(* Logix 5000 project; controller reports 1756-L63 rev 20.11; software revision 20.04; part 2 of 52 *)

        [93].log_data[7].valid := 1, [93].log_data[8].valid := 1, [93].log_data[9].valid := 1, [93].log_data[10].valid := 1, [93].log_data[11].valid := 1, [93].log_data[12].valid := 1, [93].log_data[13].valid := 1, [93].log_data[14].valid := 1, [93].log_data[15].valid := 1, [93].log_data[16].valid := 1, [93].log_data[17].valid := 1, [93].log_data[18].valid := 1, [93].log_data[19].valid := 1, [93].time.Year := 2023, [93].time.Month := 1, [93].time.Day := 16, [93].time.Hour := 23, [93].time.Minute := 44, [93].time.Second := 59, [94].log_data[0].min := 1.0, [94].log_data[0].max := 1.0, [94].log_data[0].total := 900.0, [94].log_data[0].time := 900.0, [94].log_data[0].minminute := 45, [94].log_data[0].maxminute := 45, [94].log_data[0].valid := 1, [94].log_data[1].valid := 1, [94].log_data[2].valid := 1, [94].log_data[3].valid := 1, [94].log_data[4].valid := 1, [94].log_data[5].valid := 1, [94].log_data[6].valid := 1, [94].log_data[7].valid := 1, [94].log_data[8].valid := 1, [94].log_data[9].valid := 1, [94].log_data[10].valid := 1, [94].log_data[11].valid := 1, [94].log_data[12].valid := 1, [94].log_data[13].valid := 1, [94].log_data[14].valid := 1, [94].log_data[15].valid := 1, [94].log_data[16].valid := 1, [94].log_data[17].valid := 1, [94].log_data[18].valid := 1, [94].log_data[19].valid := 1, [94].time.Year := 2023, [94].time.Month := 1, [94].time.Day := 16, [94].time.Hour := 23, [94].time.Minute := 59, [94].time.Second := 59, [95].log_data[0].min := 1.0, [95].log_data[0].max := 1.0, [95].log_data[0].total := 900.0, [95].log_data[0].time := 900.0, [95].log_data[0].valid := 1, [95].log_data[1].valid := 1, [95].log_data[2].valid := 1, [95].log_data[3].valid := 1, [95].log_data[4].valid := 1,
        [95].log_data[5].valid := 1, [95].log_data[6].valid := 1, [95].log_data[7].valid := 1, [95].log_data[8].valid := 1, [95].log_data[9].valid := 1, [95].log_data[10].valid := 1, [95].log_data[11].valid := 1, [95].log_data[12].valid := 1, [95].log_data[13].valid := 1, [95].log_data[14].valid := 1, [95].log_data[15].valid := 1, [95].log_data[16].valid := 1, [95].log_data[17].valid := 1, [95].log_data[18].valid := 1, [95].log_data[19].valid := 1, [95].time.Year := 2023, [95].time.Month := 1, [95].time.Day := 17, [95].time.Minute := 14, [95].time.Second := 59, [96].log_data[0].min := 1.0, [96].log_data[0].max := 1.0, [96].log_data[0].total := 900.0, [96].log_data[0].time := 900.0, [96].log_data[0].minminute := 15, [96].log_data[0].maxminute := 15, [96].log_data[0].valid := 1, [96].log_data[1].valid := 1, [96].log_data[2].valid := 1, [96].log_data[3].valid := 1, [96].log_data[4].valid := 1, [96].log_data[5].valid := 1, [96].log_data[6].valid := 1, [96].log_data[7].valid := 1, [96].log_data[8].valid := 1, [96].log_data[9].valid := 1, [96].log_data[10].valid := 1, [96].log_data[11].valid := 1, [96].log_data[12].valid := 1, [96].log_data[13].valid := 1, [96].log_data[14].valid := 1, [96].log_data[15].valid := 1, [96].log_data[16].valid := 1, [96].log_data[17].valid := 1, [96].log_data[18].valid := 1, [96].log_data[19].valid := 1, [96].time.Year := 2023, [96].time.Month := 1, [96].time.Day := 17, [96].time.Minute := 29, [96].time.Second := 59, [97].log_data[0].min := 1.0, [97].log_data[0].max := 1.0, [97].log_data[0].total := 900.0, [97].log_data[0].time := 900.0, [97].log_data[0].minminute := 30, [97].log_data[0].maxminute := 30, [97].log_data[0].valid := 1, [97].log_data[1].valid := 1, [97].log_data[2].valid := 1,
        [97].log_data[3].valid := 1, [97].log_data[4].valid := 1, [97].log_data[5].valid := 1, [97].log_data[6].valid := 1, [97].log_data[7].valid := 1, [97].log_data[8].valid := 1, [97].log_data[9].valid := 1, [97].log_data[10].valid := 1, [97].log_data[11].valid := 1, [97].log_data[12].valid := 1, [97].log_data[13].valid := 1, [97].log_data[14].valid := 1, [97].log_data[15].valid := 1, [97].log_data[16].valid := 1, [97].log_data[17].valid := 1, [97].log_data[18].valid := 1, [97].log_data[19].valid := 1, [97].time.Year := 2023, [97].time.Month := 1, [97].time.Day := 17, [97].time.Minute := 44, [97].time.Second := 59, [98].log_data[0].min := 1.0, [98].log_data[0].max := 1.0, [98].log_data[0].total := 900.0, [98].log_data[0].time := 900.0, [98].log_data[0].minminute := 45, [98].log_data[0].maxminute := 45, [98].log_data[0].valid := 1, [98].log_data[1].valid := 1, [98].log_data[2].valid := 1, [98].log_data[3].valid := 1, [98].log_data[4].valid := 1, [98].log_data[5].valid := 1, [98].log_data[6].valid := 1, [98].log_data[7].valid := 1, [98].log_data[8].valid := 1, [98].log_data[9].valid := 1, [98].log_data[10].valid := 1, [98].log_data[11].valid := 1, [98].log_data[12].valid := 1, [98].log_data[13].valid := 1, [98].log_data[14].valid := 1, [98].log_data[15].valid := 1, [98].log_data[16].valid := 1, [98].log_data[17].valid := 1, [98].log_data[18].valid := 1, [98].log_data[19].valid := 1, [98].time.Year := 2023, [98].time.Month := 1, [98].time.Day := 17, [98].time.Minute := 59, [98].time.Second := 59, [99].log_data[0].min := 1.0, [99].log_data[0].max := 1.0, [99].log_data[0].total := 900.0, [99].log_data[0].time := 900.0, [99].log_data[0].valid := 1, [99].log_data[1].valid := 1, [99].log_data[2].valid := 1,
        [99].log_data[3].valid := 1, [99].log_data[4].valid := 1, [99].log_data[5].valid := 1, [99].log_data[6].valid := 1, [99].log_data[7].valid := 1, [99].log_data[8].valid := 1, [99].log_data[9].valid := 1, [99].log_data[10].valid := 1, [99].log_data[11].valid := 1, [99].log_data[12].valid := 1, [99].log_data[13].valid := 1, [99].log_data[14].valid := 1, [99].log_data[15].valid := 1, [99].log_data[16].valid := 1, [99].log_data[17].valid := 1, [99].log_data[18].valid := 1, [99].log_data[19].valid := 1, [99].time.Year := 2023, [99].time.Month := 1, [99].time.Day := 17, [99].time.Hour := 1, [99].time.Minute := 14, [99].time.Second := 59, [100].log_data[0].min := 1.0, [100].log_data[0].max := 1.0, [100].log_data[0].total := 900.0, [100].log_data[0].time := 900.0, [100].log_data[0].minminute := 15, [100].log_data[0].maxminute := 15, [100].log_data[0].valid := 1, [100].log_data[1].valid := 1, [100].log_data[2].valid := 1, [100].log_data[3].valid := 1, [100].log_data[4].valid := 1, [100].log_data[5].valid := 1, [100].log_data[6].valid := 1, [100].log_data[7].valid := 1, [100].log_data[8].valid := 1, [100].log_data[9].valid := 1, [100].log_data[10].valid := 1, [100].log_data[11].valid := 1, [100].log_data[12].valid := 1, [100].log_data[13].valid := 1, [100].log_data[14].valid := 1, [100].log_data[15].valid := 1, [100].log_data[16].valid := 1, [100].log_data[17].valid := 1, [100].log_data[18].valid := 1, [100].log_data[19].valid := 1, [100].time.Year := 2023, [100].time.Month := 1, [100].time.Day := 17, [100].time.Hour := 1, [100].time.Minute := 29, [100].time.Second := 59, [101].log_data[0].min := 1.0, [101].log_data[0].max := 1.0, [101].log_data[0].total := 900.0, [101].log_data[0].time := 900.0, [101].log_data[0].minminute := 30,
        [101].log_data[0].maxminute := 30, [101].log_data[0].valid := 1, [101].log_data[1].valid := 1, [101].log_data[2].valid := 1, [101].log_data[3].valid := 1, [101].log_data[4].valid := 1, [101].log_data[5].valid := 1, [101].log_data[6].valid := 1, [101].log_data[7].valid := 1, [101].log_data[8].valid := 1, [101].log_data[9].valid := 1, [101].log_data[10].valid := 1, [101].log_data[11].valid := 1, [101].log_data[12].valid := 1, [101].log_data[13].valid := 1, [101].log_data[14].valid := 1, [101].log_data[15].valid := 1, [101].log_data[16].valid := 1, [101].log_data[17].valid := 1, [101].log_data[18].valid := 1, [101].log_data[19].valid := 1, [101].time.Year := 2023, [101].time.Month := 1, [101].time.Day := 17, [101].time.Hour := 1, [101].time.Minute := 44, [101].time.Second := 59, [102].log_data[0].min := 1.0, [102].log_data[0].max := 1.0, [102].log_data[0].total := 900.0, [102].log_data[0].time := 900.0, [102].log_data[0].minminute := 45, [102].log_data[0].maxminute := 45, [102].log_data[0].valid := 1, [102].log_data[1].valid := 1, [102].log_data[2].valid := 1, [102].log_data[3].valid := 1, [102].log_data[4].valid := 1, [102].log_data[5].valid := 1, [102].log_data[6].valid := 1, [102].log_data[7].valid := 1, [102].log_data[8].valid := 1, [102].log_data[9].valid := 1, [102].log_data[10].valid := 1, [102].log_data[11].valid := 1, [102].log_data[12].valid := 1, [102].log_data[13].valid := 1, [102].log_data[14].valid := 1, [102].log_data[15].valid := 1, [102].log_data[16].valid := 1, [102].log_data[17].valid := 1, [102].log_data[18].valid := 1, [102].log_data[19].valid := 1, [102].time.Year := 2023, [102].time.Month := 1, [102].time.Day := 17, [102].time.Hour := 1, [102].time.Minute := 59, [102].time.Second := 59, [103].log_data[0].min := 1.0,
        [103].log_data[0].max := 1.0, [103].log_data[0].total := 900.0, [103].log_data[0].time := 900.0, [103].log_data[0].valid := 1, [103].log_data[1].valid := 1, [103].log_data[2].valid := 1, [103].log_data[3].valid := 1, [103].log_data[4].valid := 1, [103].log_data[5].valid := 1, [103].log_data[6].valid := 1, [103].log_data[7].valid := 1, [103].log_data[8].valid := 1, [103].log_data[9].valid := 1, [103].log_data[10].valid := 1, [103].log_data[11].valid := 1, [103].log_data[12].valid := 1, [103].log_data[13].valid := 1, [103].log_data[14].valid := 1, [103].log_data[15].valid := 1, [103].log_data[16].valid := 1, [103].log_data[17].valid := 1, [103].log_data[18].valid := 1, [103].log_data[19].valid := 1, [103].time.Year := 2023, [103].time.Month := 1, [103].time.Day := 17, [103].time.Hour := 2, [103].time.Minute := 14, [103].time.Second := 59, [104].log_data[0].min := 1.0, [104].log_data[0].max := 1.0, [104].log_data[0].total := 900.0, [104].log_data[0].time := 900.0, [104].log_data[0].minminute := 15, [104].log_data[0].maxminute := 15, [104].log_data[0].valid := 1, [104].log_data[1].valid := 1, [104].log_data[2].valid := 1, [104].log_data[3].valid := 1, [104].log_data[4].valid := 1, [104].log_data[5].valid := 1, [104].log_data[6].valid := 1, [104].log_data[7].valid := 1, [104].log_data[8].valid := 1, [104].log_data[9].valid := 1, [104].log_data[10].valid := 1, [104].log_data[11].valid := 1, [104].log_data[12].valid := 1, [104].log_data[13].valid := 1, [104].log_data[14].valid := 1, [104].log_data[15].valid := 1, [104].log_data[16].valid := 1, [104].log_data[17].valid := 1, [104].log_data[18].valid := 1, [104].log_data[19].valid := 1, [104].time.Year := 2023, [104].time.Month := 1, [104].time.Day := 17, [104].time.Hour := 2, [104].time.Minute := 29,
        [104].time.Second := 59, [105].log_data[0].min := 1.0, [105].log_data[0].max := 1.0, [105].log_data[0].total := 900.0, [105].log_data[0].time := 900.0, [105].log_data[0].minminute := 30, [105].log_data[0].maxminute := 30, [105].log_data[0].valid := 1, [105].log_data[1].valid := 1, [105].log_data[2].valid := 1, [105].log_data[3].valid := 1, [105].log_data[4].valid := 1, [105].log_data[5].valid := 1, [105].log_data[6].valid := 1, [105].log_data[7].valid := 1, [105].log_data[8].valid := 1, [105].log_data[9].valid := 1, [105].log_data[10].valid := 1, [105].log_data[11].valid := 1, [105].log_data[12].valid := 1, [105].log_data[13].valid := 1, [105].log_data[14].valid := 1, [105].log_data[15].valid := 1, [105].log_data[16].valid := 1, [105].log_data[17].valid := 1, [105].log_data[18].valid := 1, [105].log_data[19].valid := 1, [105].time.Year := 2023, [105].time.Month := 1, [105].time.Day := 17, [105].time.Hour := 2, [105].time.Minute := 44, [105].time.Second := 59, [106].log_data[0].min := 1.0, [106].log_data[0].max := 1.0, [106].log_data[0].total := 900.0, [106].log_data[0].time := 900.0, [106].log_data[0].minminute := 45, [106].log_data[0].maxminute := 45, [106].log_data[0].valid := 1, [106].log_data[1].valid := 1, [106].log_data[2].valid := 1, [106].log_data[3].valid := 1, [106].log_data[4].valid := 1, [106].log_data[5].valid := 1, [106].log_data[6].valid := 1, [106].log_data[7].valid := 1, [106].log_data[8].valid := 1, [106].log_data[9].valid := 1, [106].log_data[10].valid := 1, [106].log_data[11].valid := 1, [106].log_data[12].valid := 1, [106].log_data[13].valid := 1, [106].log_data[14].valid := 1, [106].log_data[15].valid := 1, [106].log_data[16].valid := 1, [106].log_data[17].valid := 1, [106].log_data[18].valid := 1, [106].log_data[19].valid := 1, [106].time.Year := 2023,
        [106].time.Month := 1, [106].time.Day := 17, [106].time.Hour := 2, [106].time.Minute := 59, [106].time.Second := 59, [107].log_data[0].min := 1.0, [107].log_data[0].max := 1.0, [107].log_data[0].total := 900.0, [107].log_data[0].time := 900.0, [107].log_data[0].valid := 1, [107].log_data[1].valid := 1, [107].log_data[2].valid := 1, [107].log_data[3].valid := 1, [107].log_data[4].valid := 1, [107].log_data[5].valid := 1, [107].log_data[6].valid := 1, [107].log_data[7].valid := 1, [107].log_data[8].valid := 1, [107].log_data[9].valid := 1, [107].log_data[10].valid := 1, [107].log_data[11].valid := 1, [107].log_data[12].valid := 1, [107].log_data[13].valid := 1, [107].log_data[14].valid := 1, [107].log_data[15].valid := 1, [107].log_data[16].valid := 1, [107].log_data[17].valid := 1, [107].log_data[18].valid := 1, [107].log_data[19].valid := 1, [107].time.Year := 2023, [107].time.Month := 1, [107].time.Day := 17, [107].time.Hour := 3, [107].time.Minute := 14, [107].time.Second := 59, [108].log_data[0].min := 1.0, [108].log_data[0].max := 1.0, [108].log_data[0].total := 900.0, [108].log_data[0].time := 900.0, [108].log_data[0].minminute := 15, [108].log_data[0].maxminute := 15, [108].log_data[0].valid := 1, [108].log_data[1].valid := 1, [108].log_data[2].valid := 1, [108].log_data[3].valid := 1, [108].log_data[4].valid := 1, [108].log_data[5].valid := 1, [108].log_data[6].valid := 1, [108].log_data[7].valid := 1, [108].log_data[8].valid := 1, [108].log_data[9].valid := 1, [108].log_data[10].valid := 1, [108].log_data[11].valid := 1, [108].log_data[12].valid := 1, [108].log_data[13].valid := 1, [108].log_data[14].valid := 1, [108].log_data[15].valid := 1, [108].log_data[16].valid := 1, [108].log_data[17].valid := 1, [108].log_data[18].valid := 1,
        [108].log_data[19].valid := 1, [108].time.Year := 2023, [108].time.Month := 1, [108].time.Day := 17, [108].time.Hour := 3, [108].time.Minute := 29, [108].time.Second := 59, [109].log_data[0].min := 1.0, [109].log_data[0].max := 1.0, [109].log_data[0].total := 900.0, [109].log_data[0].time := 900.0, [109].log_data[0].minminute := 30, [109].log_data[0].maxminute := 30, [109].log_data[0].valid := 1, [109].log_data[1].valid := 1, [109].log_data[2].valid := 1, [109].log_data[3].valid := 1, [109].log_data[4].valid := 1, [109].log_data[5].valid := 1, [109].log_data[6].valid := 1, [109].log_data[7].valid := 1, [109].log_data[8].valid := 1, [109].log_data[9].valid := 1, [109].log_data[10].valid := 1, [109].log_data[11].valid := 1, [109].log_data[12].valid := 1, [109].log_data[13].valid := 1, [109].log_data[14].valid := 1, [109].log_data[15].valid := 1, [109].log_data[16].valid := 1, [109].log_data[17].valid := 1, [109].log_data[18].valid := 1, [109].log_data[19].valid := 1, [109].time.Year := 2023, [109].time.Month := 1, [109].time.Day := 17, [109].time.Hour := 3, [109].time.Minute := 44, [109].time.Second := 59, [110].log_data[0].min := 1.0, [110].log_data[0].max := 1.0, [110].log_data[0].total := 900.0, [110].log_data[0].time := 900.0, [110].log_data[0].minminute := 45, [110].log_data[0].maxminute := 45, [110].log_data[0].valid := 1, [110].log_data[1].valid := 1, [110].log_data[2].valid := 1, [110].log_data[3].valid := 1, [110].log_data[4].valid := 1, [110].log_data[5].valid := 1, [110].log_data[6].valid := 1, [110].log_data[7].valid := 1, [110].log_data[8].valid := 1, [110].log_data[9].valid := 1, [110].log_data[10].valid := 1, [110].log_data[11].valid := 1, [110].log_data[12].valid := 1, [110].log_data[13].valid := 1, [110].log_data[14].valid := 1,
        [110].log_data[15].valid := 1, [110].log_data[16].valid := 1, [110].log_data[17].valid := 1, [110].log_data[18].valid := 1, [110].log_data[19].valid := 1, [110].time.Year := 2023, [110].time.Month := 1, [110].time.Day := 17, [110].time.Hour := 3, [110].time.Minute := 59, [110].time.Second := 59, [111].log_data[0].min := 1.0, [111].log_data[0].max := 1.0, [111].log_data[0].total := 900.0, [111].log_data[0].time := 900.0, [111].log_data[0].valid := 1, [111].log_data[1].valid := 1, [111].log_data[2].valid := 1, [111].log_data[3].valid := 1, [111].log_data[4].valid := 1, [111].log_data[5].valid := 1, [111].log_data[6].valid := 1, [111].log_data[7].valid := 1, [111].log_data[8].valid := 1, [111].log_data[9].valid := 1, [111].log_data[10].valid := 1, [111].log_data[11].valid := 1, [111].log_data[12].valid := 1, [111].log_data[13].valid := 1, [111].log_data[14].valid := 1, [111].log_data[15].valid := 1, [111].log_data[16].valid := 1, [111].log_data[17].valid := 1, [111].log_data[18].valid := 1, [111].log_data[19].valid := 1, [111].time.Year := 2023, [111].time.Month := 1, [111].time.Day := 17, [111].time.Hour := 4, [111].time.Minute := 14, [111].time.Second := 59, [112].log_data[0].min := 1.0, [112].log_data[0].max := 1.0, [112].log_data[0].total := 900.0, [112].log_data[0].time := 900.0, [112].log_data[0].minminute := 15, [112].log_data[0].maxminute := 15, [112].log_data[0].valid := 1, [112].log_data[1].valid := 1, [112].log_data[2].valid := 1, [112].log_data[3].valid := 1, [112].log_data[4].valid := 1, [112].log_data[5].valid := 1, [112].log_data[6].valid := 1, [112].log_data[7].valid := 1, [112].log_data[8].valid := 1, [112].log_data[9].valid := 1, [112].log_data[10].valid := 1, [112].log_data[11].valid := 1, [112].log_data[12].valid := 1,
        [112].log_data[13].valid := 1, [112].log_data[14].valid := 1, [112].log_data[15].valid := 1, [112].log_data[16].valid := 1, [112].log_data[17].valid := 1, [112].log_data[18].valid := 1, [112].log_data[19].valid := 1, [112].time.Year := 2023, [112].time.Month := 1, [112].time.Day := 17, [112].time.Hour := 4, [112].time.Minute := 29, [112].time.Second := 59, [113].log_data[0].min := 1.0, [113].log_data[0].max := 1.0, [113].log_data[0].total := 900.0, [113].log_data[0].time := 900.0, [113].log_data[0].minminute := 30, [113].log_data[0].maxminute := 30, [113].log_data[0].valid := 1, [113].log_data[1].valid := 1, [113].log_data[2].valid := 1, [113].log_data[3].valid := 1, [113].log_data[4].valid := 1, [113].log_data[5].valid := 1, [113].log_data[6].valid := 1, [113].log_data[7].valid := 1, [113].log_data[8].valid := 1, [113].log_data[9].valid := 1, [113].log_data[10].valid := 1, [113].log_data[11].valid := 1, [113].log_data[12].valid := 1, [113].log_data[13].valid := 1, [113].log_data[14].valid := 1, [113].log_data[15].valid := 1, [113].log_data[16].valid := 1, [113].log_data[17].valid := 1, [113].log_data[18].valid := 1, [113].log_data[19].valid := 1, [113].time.Year := 2023, [113].time.Month := 1, [113].time.Day := 17, [113].time.Hour := 4, [113].time.Minute := 44, [113].time.Second := 59, [114].log_data[0].min := 1.0, [114].log_data[0].max := 1.0, [114].log_data[0].total := 900.0, [114].log_data[0].time := 900.0, [114].log_data[0].minminute := 45, [114].log_data[0].maxminute := 45, [114].log_data[0].valid := 1, [114].log_data[1].valid := 1, [114].log_data[2].valid := 1, [114].log_data[3].valid := 1, [114].log_data[4].valid := 1, [114].log_data[5].valid := 1, [114].log_data[6].valid := 1, [114].log_data[7].valid := 1, [114].log_data[8].valid := 1,
        [114].log_data[9].valid := 1, [114].log_data[10].valid := 1, [114].log_data[11].valid := 1, [114].log_data[12].valid := 1, [114].log_data[13].valid := 1, [114].log_data[14].valid := 1, [114].log_data[15].valid := 1, [114].log_data[16].valid := 1, [114].log_data[17].valid := 1, [114].log_data[18].valid := 1, [114].log_data[19].valid := 1, [114].time.Year := 2023, [114].time.Month := 1, [114].time.Day := 17, [114].time.Hour := 4, [114].time.Minute := 59, [114].time.Second := 59, [115].log_data[0].min := 1.0, [115].log_data[0].max := 1.0, [115].log_data[0].total := 900.0, [115].log_data[0].time := 900.0, [115].log_data[0].valid := 1, [115].log_data[1].valid := 1, [115].log_data[2].valid := 1, [115].log_data[3].valid := 1, [115].log_data[4].valid := 1, [115].log_data[5].valid := 1, [115].log_data[6].valid := 1, [115].log_data[7].valid := 1, [115].log_data[8].valid := 1, [115].log_data[9].valid := 1, [115].log_data[10].valid := 1, [115].log_data[11].valid := 1, [115].log_data[12].valid := 1, [115].log_data[13].valid := 1, [115].log_data[14].valid := 1, [115].log_data[15].valid := 1, [115].log_data[16].valid := 1, [115].log_data[17].valid := 1, [115].log_data[18].valid := 1, [115].log_data[19].valid := 1, [115].time.Year := 2023, [115].time.Month := 1, [115].time.Day := 17, [115].time.Hour := 5, [115].time.Minute := 14, [115].time.Second := 59, [116].log_data[0].min := 1.0, [116].log_data[0].max := 1.0, [116].log_data[0].total := 900.0, [116].log_data[0].time := 900.0, [116].log_data[0].minminute := 15, [116].log_data[0].maxminute := 15, [116].log_data[0].valid := 1, [116].log_data[1].valid := 1, [116].log_data[2].valid := 1, [116].log_data[3].valid := 1, [116].log_data[4].valid := 1, [116].log_data[5].valid := 1, [116].log_data[6].valid := 1,
        [116].log_data[7].valid := 1, [116].log_data[8].valid := 1, [116].log_data[9].valid := 1, [116].log_data[10].valid := 1, [116].log_data[11].valid := 1, [116].log_data[12].valid := 1, [116].log_data[13].valid := 1, [116].log_data[14].valid := 1, [116].log_data[15].valid := 1, [116].log_data[16].valid := 1, [116].log_data[17].valid := 1, [116].log_data[18].valid := 1, [116].log_data[19].valid := 1, [116].time.Year := 2023, [116].time.Month := 1, [116].time.Day := 17, [116].time.Hour := 5, [116].time.Minute := 29, [116].time.Second := 59, [117].log_data[0].min := 1.0, [117].log_data[0].max := 1.0, [117].log_data[0].total := 900.0, [117].log_data[0].time := 900.0, [117].log_data[0].minminute := 30, [117].log_data[0].maxminute := 30, [117].log_data[0].valid := 1, [117].log_data[1].valid := 1, [117].log_data[2].valid := 1, [117].log_data[3].valid := 1, [117].log_data[4].valid := 1, [117].log_data[5].valid := 1, [117].log_data[6].valid := 1, [117].log_data[7].valid := 1, [117].log_data[8].valid := 1, [117].log_data[9].valid := 1, [117].log_data[10].valid := 1, [117].log_data[11].valid := 1, [117].log_data[12].valid := 1, [117].log_data[13].valid := 1, [117].log_data[14].valid := 1, [117].log_data[15].valid := 1, [117].log_data[16].valid := 1, [117].log_data[17].valid := 1, [117].log_data[18].valid := 1, [117].log_data[19].valid := 1, [117].time.Year := 2023, [117].time.Month := 1, [117].time.Day := 17, [117].time.Hour := 5, [117].time.Minute := 44, [117].time.Second := 59, [118].log_data[0].min := 1.0, [118].log_data[0].max := 1.0, [118].log_data[0].total := 900.0, [118].log_data[0].time := 900.0, [118].log_data[0].minminute := 45, [118].log_data[0].maxminute := 45, [118].log_data[0].valid := 1, [118].log_data[1].valid := 1, [118].log_data[2].valid := 1,
        [118].log_data[3].valid := 1, [118].log_data[4].valid := 1, [118].log_data[5].valid := 1, [118].log_data[6].valid := 1, [118].log_data[7].valid := 1, [118].log_data[8].valid := 1, [118].log_data[9].valid := 1, [118].log_data[10].valid := 1, [118].log_data[11].valid := 1, [118].log_data[12].valid := 1, [118].log_data[13].valid := 1, [118].log_data[14].valid := 1, [118].log_data[15].valid := 1, [118].log_data[16].valid := 1, [118].log_data[17].valid := 1, [118].log_data[18].valid := 1, [118].log_data[19].valid := 1, [118].time.Year := 2023, [118].time.Month := 1, [118].time.Day := 17, [118].time.Hour := 5, [118].time.Minute := 59, [118].time.Second := 59, [119].log_data[0].min := 1.0, [119].log_data[0].max := 1.0, [119].log_data[0].total := 900.0, [119].log_data[0].time := 900.0, [119].log_data[0].valid := 1, [119].log_data[1].valid := 1, [119].log_data[2].valid := 1, [119].log_data[3].valid := 1, [119].log_data[4].valid := 1, [119].log_data[5].valid := 1, [119].log_data[6].valid := 1, [119].log_data[7].valid := 1, [119].log_data[8].valid := 1, [119].log_data[9].valid := 1, [119].log_data[10].valid := 1, [119].log_data[11].valid := 1, [119].log_data[12].valid := 1, [119].log_data[13].valid := 1, [119].log_data[14].valid := 1, [119].log_data[15].valid := 1, [119].log_data[16].valid := 1, [119].log_data[17].valid := 1, [119].log_data[18].valid := 1, [119].log_data[19].valid := 1, [119].time.Year := 2023, [119].time.Month := 1, [119].time.Day := 17, [119].time.Hour := 6, [119].time.Minute := 14, [119].time.Second := 59, [120].log_data[0].min := 1.0, [120].log_data[0].max := 1.0, [120].log_data[0].total := 900.0, [120].log_data[0].time := 900.0, [120].log_data[0].minminute := 15, [120].log_data[0].maxminute := 15, [120].log_data[0].valid := 1,
        [120].log_data[1].valid := 1, [120].log_data[2].valid := 1, [120].log_data[3].valid := 1, [120].log_data[4].valid := 1, [120].log_data[5].valid := 1, [120].log_data[6].valid := 1, [120].log_data[7].valid := 1, [120].log_data[8].valid := 1, [120].log_data[9].valid := 1, [120].log_data[10].valid := 1, [120].log_data[11].valid := 1, [120].log_data[12].valid := 1, [120].log_data[13].valid := 1, [120].log_data[14].valid := 1, [120].log_data[15].valid := 1, [120].log_data[16].valid := 1, [120].log_data[17].valid := 1, [120].log_data[18].valid := 1, [120].log_data[19].valid := 1, [120].time.Year := 2023, [120].time.Month := 1, [120].time.Day := 17, [120].time.Hour := 6, [120].time.Minute := 29, [120].time.Second := 59, [121].log_data[0].min := 1.0, [121].log_data[0].max := 1.0, [121].log_data[0].total := 900.0, [121].log_data[0].time := 900.0, [121].log_data[0].minminute := 30, [121].log_data[0].maxminute := 30, [121].log_data[0].valid := 1, [121].log_data[1].valid := 1, [121].log_data[2].valid := 1, [121].log_data[3].valid := 1, [121].log_data[4].valid := 1, [121].log_data[5].valid := 1, [121].log_data[6].valid := 1, [121].log_data[7].valid := 1, [121].log_data[8].valid := 1, [121].log_data[9].valid := 1, [121].log_data[10].valid := 1, [121].log_data[11].valid := 1, [121].log_data[12].valid := 1, [121].log_data[13].valid := 1, [121].log_data[14].valid := 1, [121].log_data[15].valid := 1, [121].log_data[16].valid := 1, [121].log_data[17].valid := 1, [121].log_data[18].valid := 1, [121].log_data[19].valid := 1, [121].time.Year := 2023, [121].time.Month := 1, [121].time.Day := 17, [121].time.Hour := 6, [121].time.Minute := 44, [121].time.Second := 59, [122].log_data[0].min := 1.0, [122].log_data[0].max := 1.0, [122].log_data[0].total := 900.0,
        [122].log_data[0].time := 900.0, [122].log_data[0].minminute := 45, [122].log_data[0].maxminute := 45, [122].log_data[0].valid := 1, [122].log_data[1].valid := 1, [122].log_data[2].valid := 1, [122].log_data[3].valid := 1, [122].log_data[4].valid := 1, [122].log_data[5].valid := 1, [122].log_data[6].valid := 1, [122].log_data[7].valid := 1, [122].log_data[8].valid := 1, [122].log_data[9].valid := 1, [122].log_data[10].valid := 1, [122].log_data[11].valid := 1, [122].log_data[12].valid := 1, [122].log_data[13].valid := 1, [122].log_data[14].valid := 1, [122].log_data[15].valid := 1, [122].log_data[16].valid := 1, [122].log_data[17].valid := 1, [122].log_data[18].valid := 1, [122].log_data[19].valid := 1, [122].time.Year := 2023, [122].time.Month := 1, [122].time.Day := 17, [122].time.Hour := 6, [122].time.Minute := 59, [122].time.Second := 59, [123].log_data[0].min := 1.0, [123].log_data[0].max := 1.0, [123].log_data[0].total := 900.0, [123].log_data[0].time := 900.0, [123].log_data[0].valid := 1, [123].log_data[1].valid := 1, [123].log_data[2].valid := 1, [123].log_data[3].valid := 1, [123].log_data[4].valid := 1, [123].log_data[5].valid := 1, [123].log_data[6].valid := 1, [123].log_data[7].valid := 1, [123].log_data[8].valid := 1, [123].log_data[9].valid := 1, [123].log_data[10].valid := 1, [123].log_data[11].valid := 1, [123].log_data[12].valid := 1, [123].log_data[13].valid := 1, [123].log_data[14].valid := 1, [123].log_data[15].valid := 1, [123].log_data[16].valid := 1, [123].log_data[17].valid := 1, [123].log_data[18].valid := 1, [123].log_data[19].valid := 1, [123].time.Year := 2023, [123].time.Month := 1, [123].time.Day := 17, [123].time.Hour := 7, [123].time.Minute := 14, [123].time.Second := 59, [124].log_data[0].min := 1.0,
        [124].log_data[0].max := 1.0, [124].log_data[0].total := 900.0, [124].log_data[0].time := 900.0, [124].log_data[0].minminute := 15, [124].log_data[0].maxminute := 15, [124].log_data[0].valid := 1, [124].log_data[1].valid := 1, [124].log_data[2].valid := 1, [124].log_data[3].valid := 1, [124].log_data[4].valid := 1, [124].log_data[5].valid := 1, [124].log_data[6].valid := 1, [124].log_data[7].valid := 1, [124].log_data[8].valid := 1, [124].log_data[9].valid := 1, [124].log_data[10].valid := 1, [124].log_data[11].valid := 1, [124].log_data[12].valid := 1, [124].log_data[13].valid := 1, [124].log_data[14].valid := 1, [124].log_data[15].valid := 1, [124].log_data[16].valid := 1, [124].log_data[17].valid := 1, [124].log_data[18].valid := 1, [124].log_data[19].valid := 1, [124].time.Year := 2023, [124].time.Month := 1, [124].time.Day := 17, [124].time.Hour := 7, [124].time.Minute := 29, [124].time.Second := 59, [125].log_data[0].min := 1.0, [125].log_data[0].max := 1.0, [125].log_data[0].total := 900.0, [125].log_data[0].time := 900.0, [125].log_data[0].minminute := 30, [125].log_data[0].maxminute := 30, [125].log_data[0].valid := 1, [125].log_data[1].valid := 1, [125].log_data[2].valid := 1, [125].log_data[3].valid := 1, [125].log_data[4].valid := 1, [125].log_data[5].valid := 1, [125].log_data[6].valid := 1, [125].log_data[7].valid := 1, [125].log_data[8].valid := 1, [125].log_data[9].valid := 1, [125].log_data[10].valid := 1, [125].log_data[11].valid := 1, [125].log_data[12].valid := 1, [125].log_data[13].valid := 1, [125].log_data[14].valid := 1, [125].log_data[15].valid := 1, [125].log_data[16].valid := 1, [125].log_data[17].valid := 1, [125].log_data[18].valid := 1, [125].log_data[19].valid := 1, [125].time.Year := 2023, [125].time.Month := 1, [125].time.Day := 17,
        [125].time.Hour := 7, [125].time.Minute := 44, [125].time.Second := 59, [126].log_data[0].min := 1.0, [126].log_data[0].max := 1.0, [126].log_data[0].total := 900.0, [126].log_data[0].time := 900.0, [126].log_data[0].minminute := 45, [126].log_data[0].maxminute := 45, [126].log_data[0].valid := 1, [126].log_data[1].valid := 1, [126].log_data[2].valid := 1, [126].log_data[3].valid := 1, [126].log_data[4].valid := 1, [126].log_data[5].valid := 1, [126].log_data[6].valid := 1, [126].log_data[7].valid := 1, [126].log_data[8].valid := 1, [126].log_data[9].valid := 1, [126].log_data[10].valid := 1, [126].log_data[11].valid := 1, [126].log_data[12].valid := 1, [126].log_data[13].valid := 1, [126].log_data[14].valid := 1, [126].log_data[15].valid := 1, [126].log_data[16].valid := 1, [126].log_data[17].valid := 1, [126].log_data[18].valid := 1, [126].log_data[19].valid := 1, [126].time.Year := 2023, [126].time.Month := 1, [126].time.Day := 17, [126].time.Hour := 7, [126].time.Minute := 59, [126].time.Second := 59, [127].log_data[0].min := 1.0, [127].log_data[0].max := 1.0, [127].log_data[0].total := 900.0, [127].log_data[0].time := 900.0, [127].log_data[0].valid := 1, [127].log_data[1].valid := 1, [127].log_data[2].valid := 1, [127].log_data[3].valid := 1, [127].log_data[4].valid := 1, [127].log_data[5].valid := 1, [127].log_data[6].valid := 1, [127].log_data[7].valid := 1, [127].log_data[8].valid := 1, [127].log_data[9].valid := 1, [127].log_data[10].valid := 1, [127].log_data[11].valid := 1, [127].log_data[12].valid := 1, [127].log_data[13].valid := 1, [127].log_data[14].valid := 1, [127].log_data[15].valid := 1, [127].log_data[16].valid := 1, [127].log_data[17].valid := 1, [127].log_data[18].valid := 1, [127].log_data[19].valid := 1, [127].time.Year := 2023,
        [127].time.Month := 1, [127].time.Day := 17, [127].time.Hour := 8, [127].time.Minute := 14, [127].time.Second := 59, [128].log_data[0].min := 1.0, [128].log_data[0].max := 1.0, [128].log_data[0].total := 900.0, [128].log_data[0].time := 900.0, [128].log_data[0].minminute := 15, [128].log_data[0].maxminute := 15, [128].log_data[0].valid := 1, [128].log_data[1].valid := 1, [128].log_data[2].valid := 1, [128].log_data[3].valid := 1, [128].log_data[4].valid := 1, [128].log_data[5].valid := 1, [128].log_data[6].valid := 1, [128].log_data[7].valid := 1, [128].log_data[8].valid := 1, [128].log_data[9].valid := 1, [128].log_data[10].valid := 1, [128].log_data[11].valid := 1, [128].log_data[12].valid := 1, [128].log_data[13].valid := 1, [128].log_data[14].valid := 1, [128].log_data[15].valid := 1, [128].log_data[16].valid := 1, [128].log_data[17].valid := 1, [128].log_data[18].valid := 1, [128].log_data[19].valid := 1, [128].time.Year := 2023, [128].time.Month := 1, [128].time.Day := 17, [128].time.Hour := 8, [128].time.Minute := 29, [128].time.Second := 59, [129].log_data[0].min := 1.0, [129].log_data[0].max := 1.0, [129].log_data[0].total := 900.0, [129].log_data[0].time := 900.0, [129].log_data[0].minminute := 30, [129].log_data[0].maxminute := 30, [129].log_data[0].valid := 1, [129].log_data[1].valid := 1, [129].log_data[2].valid := 1, [129].log_data[3].valid := 1, [129].log_data[4].valid := 1, [129].log_data[5].valid := 1, [129].log_data[6].valid := 1, [129].log_data[7].valid := 1, [129].log_data[8].valid := 1, [129].log_data[9].valid := 1, [129].log_data[10].valid := 1, [129].log_data[11].valid := 1, [129].log_data[12].valid := 1, [129].log_data[13].valid := 1, [129].log_data[14].valid := 1, [129].log_data[15].valid := 1, [129].log_data[16].valid := 1,
        [129].log_data[17].valid := 1, [129].log_data[18].valid := 1, [129].log_data[19].valid := 1, [129].time.Year := 2023, [129].time.Month := 1, [129].time.Day := 17, [129].time.Hour := 8, [129].time.Minute := 44, [129].time.Second := 59, [130].log_data[0].min := 1.0, [130].log_data[0].max := 1.0, [130].log_data[0].total := 900.0, [130].log_data[0].time := 900.0, [130].log_data[0].minminute := 45, [130].log_data[0].maxminute := 45, [130].log_data[0].valid := 1, [130].log_data[1].valid := 1, [130].log_data[2].valid := 1, [130].log_data[3].valid := 1, [130].log_data[4].valid := 1, [130].log_data[5].valid := 1, [130].log_data[6].valid := 1, [130].log_data[7].valid := 1, [130].log_data[8].valid := 1, [130].log_data[9].valid := 1, [130].log_data[10].valid := 1, [130].log_data[11].valid := 1, [130].log_data[12].valid := 1, [130].log_data[13].valid := 1, [130].log_data[14].valid := 1, [130].log_data[15].valid := 1, [130].log_data[16].valid := 1, [130].log_data[17].valid := 1, [130].log_data[18].valid := 1, [130].log_data[19].valid := 1, [130].time.Year := 2023, [130].time.Month := 1, [130].time.Day := 17, [130].time.Hour := 8, [130].time.Minute := 59, [130].time.Second := 59, [131].log_data[0].min := 1.0, [131].log_data[0].max := 1.0, [131].log_data[0].total := 899.5, [131].log_data[0].time := 899.5, [131].log_data[0].valid := 1, [131].log_data[1].valid := 1, [131].log_data[2].valid := 1, [131].log_data[3].valid := 1, [131].log_data[4].valid := 1, [131].log_data[5].valid := 1, [131].log_data[6].valid := 1, [131].log_data[7].valid := 1, [131].log_data[8].valid := 1, [131].log_data[9].valid := 1, [131].log_data[10].valid := 1, [131].log_data[11].valid := 1, [131].log_data[12].valid := 1, [131].log_data[13].valid := 1, [131].log_data[14].valid := 1,
        [131].log_data[15].valid := 1, [131].log_data[16].valid := 1, [131].log_data[17].valid := 1, [131].log_data[18].valid := 1, [131].log_data[19].valid := 1, [131].time.Year := 2023, [131].time.Month := 1, [131].time.Day := 17, [131].time.Hour := 9, [131].time.Minute := 14, [131].time.Second := 59, [132].log_data[0].min := 1.0, [132].log_data[0].max := 1.0, [132].log_data[0].total := 900.0, [132].log_data[0].time := 900.0, [132].log_data[0].minminute := 15, [132].log_data[0].maxminute := 15, [132].log_data[0].valid := 1, [132].log_data[1].valid := 1, [132].log_data[2].valid := 1, [132].log_data[3].valid := 1, [132].log_data[4].valid := 1, [132].log_data[5].valid := 1, [132].log_data[6].valid := 1, [132].log_data[7].valid := 1, [132].log_data[8].valid := 1, [132].log_data[9].valid := 1, [132].log_data[10].valid := 1, [132].log_data[11].valid := 1, [132].log_data[12].valid := 1, [132].log_data[13].valid := 1, [132].log_data[14].valid := 1, [132].log_data[15].valid := 1, [132].log_data[16].valid := 1, [132].log_data[17].valid := 1, [132].log_data[18].valid := 1, [132].log_data[19].valid := 1, [132].time.Year := 2023, [132].time.Month := 1, [132].time.Day := 17, [132].time.Hour := 9, [132].time.Minute := 29, [132].time.Second := 59, [133].log_data[0].min := 1.0, [133].log_data[0].max := 1.0, [133].log_data[0].total := 900.0, [133].log_data[0].time := 900.0, [133].log_data[0].minminute := 30, [133].log_data[0].maxminute := 30, [133].log_data[0].valid := 1, [133].log_data[1].valid := 1, [133].log_data[2].valid := 1, [133].log_data[3].valid := 1, [133].log_data[4].valid := 1, [133].log_data[5].valid := 1, [133].log_data[6].valid := 1, [133].log_data[7].valid := 1, [133].log_data[8].valid := 1, [133].log_data[9].valid := 1, [133].log_data[10].valid := 1,
        [133].log_data[11].valid := 1, [133].log_data[12].valid := 1, [133].log_data[13].valid := 1, [133].log_data[14].valid := 1, [133].log_data[15].valid := 1, [133].log_data[16].valid := 1, [133].log_data[17].valid := 1, [133].log_data[18].valid := 1, [133].log_data[19].valid := 1, [133].time.Year := 2023, [133].time.Month := 1, [133].time.Day := 17, [133].time.Hour := 9, [133].time.Minute := 44, [133].time.Second := 59, [134].log_data[0].min := 1.0, [134].log_data[0].max := 1.0, [134].log_data[0].total := 900.0, [134].log_data[0].time := 900.0, [134].log_data[0].minminute := 45, [134].log_data[0].maxminute := 45, [134].log_data[0].valid := 1, [134].log_data[1].valid := 1, [134].log_data[2].valid := 1, [134].log_data[3].valid := 1, [134].log_data[4].valid := 1, [134].log_data[5].valid := 1, [134].log_data[6].valid := 1, [134].log_data[7].valid := 1, [134].log_data[8].valid := 1, [134].log_data[9].valid := 1, [134].log_data[10].valid := 1, [134].log_data[11].valid := 1, [134].log_data[12].valid := 1, [134].log_data[13].valid := 1, [134].log_data[14].valid := 1, [134].log_data[15].valid := 1, [134].log_data[16].valid := 1, [134].log_data[17].valid := 1, [134].log_data[18].valid := 1, [134].log_data[19].valid := 1, [134].time.Year := 2023, [134].time.Month := 1, [134].time.Day := 17, [134].time.Hour := 9, [134].time.Minute := 59, [134].time.Second := 59, [135].log_data[0].min := 1.0, [135].log_data[0].max := 1.0, [135].log_data[0].total := 900.0, [135].log_data[0].time := 900.0, [135].log_data[0].valid := 1, [135].log_data[1].valid := 1, [135].log_data[2].valid := 1, [135].log_data[3].valid := 1, [135].log_data[4].valid := 1, [135].log_data[5].valid := 1, [135].log_data[6].valid := 1, [135].log_data[7].valid := 1, [135].log_data[8].valid := 1,
        [135].log_data[9].valid := 1, [135].log_data[10].valid := 1, [135].log_data[11].valid := 1, [135].log_data[12].valid := 1, [135].log_data[13].valid := 1, [135].log_data[14].valid := 1, [135].log_data[15].valid := 1, [135].log_data[16].valid := 1, [135].log_data[17].valid := 1, [135].log_data[18].valid := 1, [135].log_data[19].valid := 1, [135].time.Year := 2023, [135].time.Month := 1, [135].time.Day := 17, [135].time.Hour := 10, [135].time.Minute := 14, [135].time.Second := 59, [136].log_data[0].min := 1.0, [136].log_data[0].max := 1.0, [136].log_data[0].total := 900.0, [136].log_data[0].time := 900.0, [136].log_data[0].minminute := 15, [136].log_data[0].maxminute := 15, [136].log_data[0].valid := 1, [136].log_data[1].valid := 1, [136].log_data[2].valid := 1, [136].log_data[3].valid := 1, [136].log_data[4].valid := 1, [136].log_data[5].valid := 1, [136].log_data[6].valid := 1, [136].log_data[7].valid := 1, [136].log_data[8].valid := 1, [136].log_data[9].valid := 1, [136].log_data[10].valid := 1, [136].log_data[11].valid := 1, [136].log_data[12].valid := 1, [136].log_data[13].valid := 1, [136].log_data[14].valid := 1, [136].log_data[15].valid := 1, [136].log_data[16].valid := 1, [136].log_data[17].valid := 1, [136].log_data[18].valid := 1, [136].log_data[19].valid := 1, [136].time.Year := 2023, [136].time.Month := 1, [136].time.Day := 17, [136].time.Hour := 10, [136].time.Minute := 29, [136].time.Second := 59, [137].log_data[0].min := 1.0, [137].log_data[0].max := 1.0, [137].log_data[0].total := 900.0, [137].log_data[0].time := 900.0, [137].log_data[0].minminute := 30, [137].log_data[0].maxminute := 30, [137].log_data[0].valid := 1, [137].log_data[1].valid := 1, [137].log_data[2].valid := 1, [137].log_data[3].valid := 1, [137].log_data[4].valid := 1,
        [137].log_data[5].valid := 1, [137].log_data[6].valid := 1, [137].log_data[7].valid := 1, [137].log_data[8].valid := 1, [137].log_data[9].valid := 1, [137].log_data[10].valid := 1, [137].log_data[11].valid := 1, [137].log_data[12].valid := 1, [137].log_data[13].valid := 1, [137].log_data[14].valid := 1, [137].log_data[15].valid := 1, [137].log_data[16].valid := 1, [137].log_data[17].valid := 1, [137].log_data[18].valid := 1, [137].log_data[19].valid := 1, [137].time.Year := 2023, [137].time.Month := 1, [137].time.Day := 17, [137].time.Hour := 10, [137].time.Minute := 44, [137].time.Second := 59, [138].log_data[0].min := 1.0, [138].log_data[0].max := 1.0, [138].log_data[0].total := 900.0, [138].log_data[0].time := 900.0, [138].log_data[0].minminute := 45, [138].log_data[0].maxminute := 45, [138].log_data[0].valid := 1, [138].log_data[1].valid := 1, [138].log_data[2].valid := 1, [138].log_data[3].valid := 1, [138].log_data[4].valid := 1, [138].log_data[5].valid := 1, [138].log_data[6].valid := 1, [138].log_data[7].valid := 1, [138].log_data[8].valid := 1, [138].log_data[9].valid := 1, [138].log_data[10].valid := 1, [138].log_data[11].valid := 1, [138].log_data[12].valid := 1, [138].log_data[13].valid := 1, [138].log_data[14].valid := 1, [138].log_data[15].valid := 1, [138].log_data[16].valid := 1, [138].log_data[17].valid := 1, [138].log_data[18].valid := 1, [138].log_data[19].valid := 1, [138].time.Year := 2023, [138].time.Month := 1, [138].time.Day := 17, [138].time.Hour := 10, [138].time.Minute := 59, [138].time.Second := 59, [139].log_data[0].min := 1.0, [139].log_data[0].max := 1.0, [139].log_data[0].total := 900.0, [139].log_data[0].time := 900.0, [139].log_data[0].valid := 1, [139].log_data[1].valid := 1, [139].log_data[2].valid := 1,
        [139].log_data[3].valid := 1, [139].log_data[4].valid := 1, [139].log_data[5].valid := 1, [139].log_data[6].valid := 1, [139].log_data[7].valid := 1, [139].log_data[8].valid := 1, [139].log_data[9].valid := 1, [139].log_data[10].valid := 1, [139].log_data[11].valid := 1, [139].log_data[12].valid := 1, [139].log_data[13].valid := 1, [139].log_data[14].valid := 1, [139].log_data[15].valid := 1, [139].log_data[16].valid := 1, [139].log_data[17].valid := 1, [139].log_data[18].valid := 1, [139].log_data[19].valid := 1, [139].time.Year := 2023, [139].time.Month := 1, [139].time.Day := 17, [139].time.Hour := 11, [139].time.Minute := 14, [139].time.Second := 59, [140].log_data[0].min := 1.0, [140].log_data[0].max := 1.0, [140].log_data[0].total := 900.0, [140].log_data[0].time := 900.0, [140].log_data[0].minminute := 15, [140].log_data[0].maxminute := 15, [140].log_data[0].valid := 1, [140].log_data[1].valid := 1, [140].log_data[2].valid := 1, [140].log_data[3].valid := 1, [140].log_data[4].valid := 1, [140].log_data[5].valid := 1, [140].log_data[6].valid := 1, [140].log_data[7].valid := 1, [140].log_data[8].valid := 1, [140].log_data[9].valid := 1, [140].log_data[10].valid := 1, [140].log_data[11].valid := 1, [140].log_data[12].valid := 1, [140].log_data[13].valid := 1, [140].log_data[14].valid := 1, [140].log_data[15].valid := 1, [140].log_data[16].valid := 1, [140].log_data[17].valid := 1, [140].log_data[18].valid := 1, [140].log_data[19].valid := 1, [140].time.Year := 2023, [140].time.Month := 1, [140].time.Day := 17, [140].time.Hour := 11, [140].time.Minute := 29, [140].time.Second := 59, [141].log_data[0].min := 1.0, [141].log_data[0].max := 1.0, [141].log_data[0].total := 900.0, [141].log_data[0].time := 900.0, [141].log_data[0].minminute := 30,
        [141].log_data[0].maxminute := 30, [141].log_data[0].valid := 1, [141].log_data[1].valid := 1, [141].log_data[2].valid := 1, [141].log_data[3].valid := 1, [141].log_data[4].valid := 1, [141].log_data[5].valid := 1, [141].log_data[6].valid := 1, [141].log_data[7].valid := 1, [141].log_data[8].valid := 1, [141].log_data[9].valid := 1, [141].log_data[10].valid := 1, [141].log_data[11].valid := 1, [141].log_data[12].valid := 1, [141].log_data[13].valid := 1, [141].log_data[14].valid := 1, [141].log_data[15].valid := 1, [141].log_data[16].valid := 1, [141].log_data[17].valid := 1, [141].log_data[18].valid := 1, [141].log_data[19].valid := 1, [141].time.Year := 2023, [141].time.Month := 1, [141].time.Day := 17, [141].time.Hour := 11, [141].time.Minute := 44, [141].time.Second := 59, [142].log_data[0].min := 1.0, [142].log_data[0].max := 1.0, [142].log_data[0].total := 900.0, [142].log_data[0].time := 900.0, [142].log_data[0].minminute := 45, [142].log_data[0].maxminute := 45, [142].log_data[0].valid := 1, [142].log_data[1].valid := 1, [142].log_data[2].valid := 1, [142].log_data[3].valid := 1, [142].log_data[4].valid := 1, [142].log_data[5].valid := 1, [142].log_data[6].valid := 1, [142].log_data[7].valid := 1, [142].log_data[8].valid := 1, [142].log_data[9].valid := 1, [142].log_data[10].valid := 1, [142].log_data[11].valid := 1, [142].log_data[12].valid := 1, [142].log_data[13].valid := 1, [142].log_data[14].valid := 1, [142].log_data[15].valid := 1, [142].log_data[16].valid := 1, [142].log_data[17].valid := 1, [142].log_data[18].valid := 1, [142].log_data[19].valid := 1, [142].time.Year := 2023, [142].time.Month := 1, [142].time.Day := 17, [142].time.Hour := 11, [142].time.Minute := 59, [142].time.Second := 59, [143].log_data[0].min := 1.0,
        [143].log_data[0].max := 1.0, [143].log_data[0].total := 900.0, [143].log_data[0].time := 900.0, [143].log_data[0].valid := 1, [143].log_data[1].valid := 1, [143].log_data[2].valid := 1, [143].log_data[3].valid := 1, [143].log_data[4].valid := 1, [143].log_data[5].valid := 1, [143].log_data[6].valid := 1, [143].log_data[7].valid := 1, [143].log_data[8].valid := 1, [143].log_data[9].valid := 1, [143].log_data[10].valid := 1, [143].log_data[11].valid := 1, [143].log_data[12].valid := 1, [143].log_data[13].valid := 1, [143].log_data[14].valid := 1, [143].log_data[15].valid := 1, [143].log_data[16].valid := 1, [143].log_data[17].valid := 1, [143].log_data[18].valid := 1, [143].log_data[19].valid := 1, [143].time.Year := 2023, [143].time.Month := 1, [143].time.Day := 17, [143].time.Hour := 12, [143].time.Minute := 14, [143].time.Second := 59, [144].log_data[0].min := 1.0, [144].log_data[0].max := 1.0, [144].log_data[0].total := 900.0, [144].log_data[0].time := 900.0, [144].log_data[0].minminute := 15, [144].log_data[0].maxminute := 15, [144].log_data[0].valid := 1, [144].log_data[1].valid := 1, [144].log_data[2].valid := 1, [144].log_data[3].valid := 1, [144].log_data[4].valid := 1, [144].log_data[5].valid := 1, [144].log_data[6].valid := 1, [144].log_data[7].valid := 1, [144].log_data[8].valid := 1, [144].log_data[9].valid := 1, [144].log_data[10].valid := 1, [144].log_data[11].valid := 1, [144].log_data[12].valid := 1, [144].log_data[13].valid := 1, [144].log_data[14].valid := 1, [144].log_data[15].valid := 1, [144].log_data[16].valid := 1, [144].log_data[17].valid := 1, [144].log_data[18].valid := 1, [144].log_data[19].valid := 1, [144].time.Year := 2023, [144].time.Month := 1, [144].time.Day := 17, [144].time.Hour := 12, [144].time.Minute := 29,
        [144].time.Second := 59, [145].log_data[0].min := 1.0, [145].log_data[0].max := 1.0, [145].log_data[0].total := 900.0, [145].log_data[0].time := 900.0, [145].log_data[0].minminute := 30, [145].log_data[0].maxminute := 30, [145].log_data[0].valid := 1, [145].log_data[1].valid := 1, [145].log_data[2].valid := 1, [145].log_data[3].valid := 1, [145].log_data[4].valid := 1, [145].log_data[5].valid := 1, [145].log_data[6].valid := 1, [145].log_data[7].valid := 1, [145].log_data[8].valid := 1, [145].log_data[9].valid := 1, [145].log_data[10].valid := 1, [145].log_data[11].valid := 1, [145].log_data[12].valid := 1, [145].log_data[13].valid := 1, [145].log_data[14].valid := 1, [145].log_data[15].valid := 1, [145].log_data[16].valid := 1, [145].log_data[17].valid := 1, [145].log_data[18].valid := 1, [145].log_data[19].valid := 1, [145].time.Year := 2023, [145].time.Month := 1, [145].time.Day := 17, [145].time.Hour := 12, [145].time.Minute := 44, [145].time.Second := 59, [146].log_data[0].min := 1.0, [146].log_data[0].max := 1.0, [146].log_data[0].total := 900.0, [146].log_data[0].time := 900.0, [146].log_data[0].minminute := 45, [146].log_data[0].maxminute := 45, [146].log_data[0].valid := 1, [146].log_data[1].valid := 1, [146].log_data[2].valid := 1, [146].log_data[3].valid := 1, [146].log_data[4].valid := 1, [146].log_data[5].valid := 1, [146].log_data[6].valid := 1, [146].log_data[7].valid := 1, [146].log_data[8].valid := 1, [146].log_data[9].valid := 1, [146].log_data[10].valid := 1, [146].log_data[11].valid := 1, [146].log_data[12].valid := 1, [146].log_data[13].valid := 1, [146].log_data[14].valid := 1, [146].log_data[15].valid := 1, [146].log_data[16].valid := 1, [146].log_data[17].valid := 1, [146].log_data[18].valid := 1, [146].log_data[19].valid := 1, [146].time.Year := 2023,
        [146].time.Month := 1, [146].time.Day := 17, [146].time.Hour := 12, [146].time.Minute := 59, [146].time.Second := 59, [147].log_data[0].min := 1.0, [147].log_data[0].max := 1.0, [147].log_data[0].total := 900.0, [147].log_data[0].time := 900.0, [147].log_data[0].valid := 1, [147].log_data[1].valid := 1, [147].log_data[2].valid := 1, [147].log_data[3].valid := 1, [147].log_data[4].valid := 1, [147].log_data[5].valid := 1, [147].log_data[6].valid := 1, [147].log_data[7].valid := 1, [147].log_data[8].valid := 1, [147].log_data[9].valid := 1, [147].log_data[10].valid := 1, [147].log_data[11].valid := 1, [147].log_data[12].valid := 1, [147].log_data[13].valid := 1, [147].log_data[14].valid := 1, [147].log_data[15].valid := 1, [147].log_data[16].valid := 1, [147].log_data[17].valid := 1, [147].log_data[18].valid := 1, [147].log_data[19].valid := 1, [147].time.Year := 2023, [147].time.Month := 1, [147].time.Day := 17, [147].time.Hour := 13, [147].time.Minute := 14, [147].time.Second := 59, [148].log_data[0].min := 1.0, [148].log_data[0].max := 1.0, [148].log_data[0].total := 900.0, [148].log_data[0].time := 900.0, [148].log_data[0].minminute := 15, [148].log_data[0].maxminute := 15, [148].log_data[0].valid := 1, [148].log_data[1].valid := 1, [148].log_data[2].valid := 1, [148].log_data[3].valid := 1, [148].log_data[4].valid := 1, [148].log_data[5].valid := 1, [148].log_data[6].valid := 1, [148].log_data[7].valid := 1, [148].log_data[8].valid := 1, [148].log_data[9].valid := 1, [148].log_data[10].valid := 1, [148].log_data[11].valid := 1, [148].log_data[12].valid := 1, [148].log_data[13].valid := 1, [148].log_data[14].valid := 1, [148].log_data[15].valid := 1, [148].log_data[16].valid := 1, [148].log_data[17].valid := 1, [148].log_data[18].valid := 1,
        [148].log_data[19].valid := 1, [148].time.Year := 2023, [148].time.Month := 1, [148].time.Day := 17, [148].time.Hour := 13, [148].time.Minute := 29, [148].time.Second := 59, [149].log_data[0].min := 1.0, [149].log_data[0].max := 1.0, [149].log_data[0].total := 900.0, [149].log_data[0].time := 900.0, [149].log_data[0].minminute := 30, [149].log_data[0].maxminute := 30, [149].log_data[0].valid := 1, [149].log_data[1].valid := 1, [149].log_data[2].valid := 1, [149].log_data[3].valid := 1, [149].log_data[4].valid := 1, [149].log_data[5].valid := 1, [149].log_data[6].valid := 1, [149].log_data[7].valid := 1, [149].log_data[8].valid := 1, [149].log_data[9].valid := 1, [149].log_data[10].valid := 1, [149].log_data[11].valid := 1, [149].log_data[12].valid := 1, [149].log_data[13].valid := 1, [149].log_data[14].valid := 1, [149].log_data[15].valid := 1, [149].log_data[16].valid := 1, [149].log_data[17].valid := 1, [149].log_data[18].valid := 1, [149].log_data[19].valid := 1, [149].time.Year := 2023, [149].time.Month := 1, [149].time.Day := 17, [149].time.Hour := 13, [149].time.Minute := 44, [149].time.Second := 59, [150].log_data[0].min := 1.0, [150].log_data[0].max := 1.0, [150].log_data[0].total := 900.0, [150].log_data[0].time := 900.0, [150].log_data[0].minminute := 45, [150].log_data[0].maxminute := 45, [150].log_data[0].valid := 1, [150].log_data[1].valid := 1, [150].log_data[2].valid := 1, [150].log_data[3].valid := 1, [150].log_data[4].valid := 1, [150].log_data[5].valid := 1, [150].log_data[6].valid := 1, [150].log_data[7].valid := 1, [150].log_data[8].valid := 1, [150].log_data[9].valid := 1, [150].log_data[10].valid := 1, [150].log_data[11].valid := 1, [150].log_data[12].valid := 1, [150].log_data[13].valid := 1, [150].log_data[14].valid := 1,
        [150].log_data[15].valid := 1, [150].log_data[16].valid := 1, [150].log_data[17].valid := 1, [150].log_data[18].valid := 1, [150].log_data[19].valid := 1, [150].time.Year := 2023, [150].time.Month := 1, [150].time.Day := 17, [150].time.Hour := 13, [150].time.Minute := 59, [150].time.Second := 59, [151].log_data[0].min := 1.0, [151].log_data[0].max := 1.0, [151].log_data[0].total := 900.0, [151].log_data[0].time := 900.0, [151].log_data[0].valid := 1, [151].log_data[1].valid := 1, [151].log_data[2].valid := 1, [151].log_data[3].valid := 1, [151].log_data[4].valid := 1, [151].log_data[5].valid := 1, [151].log_data[6].valid := 1, [151].log_data[7].valid := 1, [151].log_data[8].valid := 1, [151].log_data[9].valid := 1, [151].log_data[10].valid := 1, [151].log_data[11].valid := 1, [151].log_data[12].valid := 1, [151].log_data[13].valid := 1, [151].log_data[14].valid := 1, [151].log_data[15].valid := 1, [151].log_data[16].valid := 1, [151].log_data[17].valid := 1, [151].log_data[18].valid := 1, [151].log_data[19].valid := 1, [151].time.Year := 2023, [151].time.Month := 1, [151].time.Day := 17, [151].time.Hour := 14, [151].time.Minute := 14, [151].time.Second := 59, [152].log_data[0].min := 1.0, [152].log_data[0].max := 1.0, [152].log_data[0].total := 900.0, [152].log_data[0].time := 900.0, [152].log_data[0].minminute := 15, [152].log_data[0].maxminute := 15, [152].log_data[0].valid := 1, [152].log_data[1].valid := 1, [152].log_data[2].valid := 1, [152].log_data[3].valid := 1, [152].log_data[4].valid := 1, [152].log_data[5].valid := 1, [152].log_data[6].valid := 1, [152].log_data[7].valid := 1, [152].log_data[8].valid := 1, [152].log_data[9].valid := 1, [152].log_data[10].valid := 1, [152].log_data[11].valid := 1, [152].log_data[12].valid := 1,
        [152].log_data[13].valid := 1, [152].log_data[14].valid := 1, [152].log_data[15].valid := 1, [152].log_data[16].valid := 1, [152].log_data[17].valid := 1, [152].log_data[18].valid := 1, [152].log_data[19].valid := 1, [152].time.Year := 2023, [152].time.Month := 1, [152].time.Day := 17, [152].time.Hour := 14, [152].time.Minute := 29, [152].time.Second := 59, [153].log_data[0].min := 1.0, [153].log_data[0].max := 1.0, [153].log_data[0].total := 900.0, [153].log_data[0].time := 900.0, [153].log_data[0].minminute := 30, [153].log_data[0].maxminute := 30, [153].log_data[0].valid := 1, [153].log_data[1].valid := 1, [153].log_data[2].valid := 1, [153].log_data[3].valid := 1, [153].log_data[4].valid := 1, [153].log_data[5].valid := 1, [153].log_data[6].valid := 1, [153].log_data[7].valid := 1, [153].log_data[8].valid := 1, [153].log_data[9].valid := 1, [153].log_data[10].valid := 1, [153].log_data[11].valid := 1, [153].log_data[12].valid := 1, [153].log_data[13].valid := 1, [153].log_data[14].valid := 1, [153].log_data[15].valid := 1, [153].log_data[16].valid := 1, [153].log_data[17].valid := 1, [153].log_data[18].valid := 1, [153].log_data[19].valid := 1, [153].time.Year := 2023, [153].time.Month := 1, [153].time.Day := 17, [153].time.Hour := 14, [153].time.Minute := 44, [153].time.Second := 59, [154].log_data[0].min := 1.0, [154].log_data[0].max := 1.0, [154].log_data[0].total := 900.0, [154].log_data[0].time := 900.0, [154].log_data[0].minminute := 45, [154].log_data[0].maxminute := 45, [154].log_data[0].valid := 1, [154].log_data[1].valid := 1, [154].log_data[2].valid := 1, [154].log_data[3].valid := 1, [154].log_data[4].valid := 1, [154].log_data[5].valid := 1, [154].log_data[6].valid := 1, [154].log_data[7].valid := 1, [154].log_data[8].valid := 1,
        [154].log_data[9].valid := 1, [154].log_data[10].valid := 1, [154].log_data[11].valid := 1, [154].log_data[12].valid := 1, [154].log_data[13].valid := 1, [154].log_data[14].valid := 1, [154].log_data[15].valid := 1, [154].log_data[16].valid := 1, [154].log_data[17].valid := 1, [154].log_data[18].valid := 1, [154].log_data[19].valid := 1, [154].time.Year := 2023, [154].time.Month := 1, [154].time.Day := 17, [154].time.Hour := 14, [154].time.Minute := 59, [154].time.Second := 59, [155].log_data[0].min := 1.0, [155].log_data[0].max := 1.0, [155].log_data[0].total := 900.0, [155].log_data[0].time := 900.0, [155].log_data[0].valid := 1, [155].log_data[1].valid := 1, [155].log_data[2].valid := 1, [155].log_data[3].valid := 1, [155].log_data[4].valid := 1, [155].log_data[5].valid := 1, [155].log_data[6].valid := 1, [155].log_data[7].valid := 1, [155].log_data[8].valid := 1, [155].log_data[9].valid := 1, [155].log_data[10].valid := 1, [155].log_data[11].valid := 1, [155].log_data[12].valid := 1, [155].log_data[13].valid := 1, [155].log_data[14].valid := 1, [155].log_data[15].valid := 1, [155].log_data[16].valid := 1, [155].log_data[17].valid := 1, [155].log_data[18].valid := 1, [155].log_data[19].valid := 1, [155].time.Year := 2023, [155].time.Month := 1, [155].time.Day := 17, [155].time.Hour := 15, [155].time.Minute := 14, [155].time.Second := 59, [156].log_data[0].min := 1.0, [156].log_data[0].max := 1.0, [156].log_data[0].total := 900.0, [156].log_data[0].time := 900.0, [156].log_data[0].minminute := 15, [156].log_data[0].maxminute := 15, [156].log_data[0].valid := 1, [156].log_data[1].valid := 1, [156].log_data[2].valid := 1, [156].log_data[3].valid := 1, [156].log_data[4].valid := 1, [156].log_data[5].valid := 1, [156].log_data[6].valid := 1,
        [156].log_data[7].valid := 1, [156].log_data[8].valid := 1, [156].log_data[9].valid := 1, [156].log_data[10].valid := 1, [156].log_data[11].valid := 1, [156].log_data[12].valid := 1, [156].log_data[13].valid := 1, [156].log_data[14].valid := 1, [156].log_data[15].valid := 1, [156].log_data[16].valid := 1, [156].log_data[17].valid := 1, [156].log_data[18].valid := 1, [156].log_data[19].valid := 1, [156].time.Year := 2023, [156].time.Month := 1, [156].time.Day := 17, [156].time.Hour := 15, [156].time.Minute := 29, [156].time.Second := 59, [157].log_data[0].min := 1.0, [157].log_data[0].max := 1.0, [157].log_data[0].total := 900.0, [157].log_data[0].time := 900.0, [157].log_data[0].minminute := 30, [157].log_data[0].maxminute := 30, [157].log_data[0].valid := 1, [157].log_data[1].valid := 1, [157].log_data[2].valid := 1, [157].log_data[3].valid := 1, [157].log_data[4].valid := 1, [157].log_data[5].valid := 1, [157].log_data[6].valid := 1, [157].log_data[7].valid := 1, [157].log_data[8].valid := 1, [157].log_data[9].valid := 1, [157].log_data[10].valid := 1, [157].log_data[11].valid := 1, [157].log_data[12].valid := 1, [157].log_data[13].valid := 1, [157].log_data[14].valid := 1, [157].log_data[15].valid := 1, [157].log_data[16].valid := 1, [157].log_data[17].valid := 1, [157].log_data[18].valid := 1, [157].log_data[19].valid := 1, [157].time.Year := 2023, [157].time.Month := 1, [157].time.Day := 17, [157].time.Hour := 15, [157].time.Minute := 44, [157].time.Second := 59, [158].log_data[0].min := 1.0, [158].log_data[0].max := 1.0, [158].log_data[0].total := 900.0, [158].log_data[0].time := 900.0, [158].log_data[0].minminute := 45, [158].log_data[0].maxminute := 45, [158].log_data[0].valid := 1, [158].log_data[1].valid := 1, [158].log_data[2].valid := 1,
        [158].log_data[3].valid := 1, [158].log_data[4].valid := 1, [158].log_data[5].valid := 1, [158].log_data[6].valid := 1, [158].log_data[7].valid := 1, [158].log_data[8].valid := 1, [158].log_data[9].valid := 1, [158].log_data[10].valid := 1, [158].log_data[11].valid := 1, [158].log_data[12].valid := 1, [158].log_data[13].valid := 1, [158].log_data[14].valid := 1, [158].log_data[15].valid := 1, [158].log_data[16].valid := 1, [158].log_data[17].valid := 1, [158].log_data[18].valid := 1, [158].log_data[19].valid := 1, [158].time.Year := 2023, [158].time.Month := 1, [158].time.Day := 17, [158].time.Hour := 15, [158].time.Minute := 59, [158].time.Second := 59, [159].log_data[0].min := 1.0, [159].log_data[0].max := 1.0, [159].log_data[0].total := 900.0, [159].log_data[0].time := 900.0, [159].log_data[0].valid := 1, [159].log_data[1].valid := 1, [159].log_data[2].valid := 1, [159].log_data[3].valid := 1, [159].log_data[4].valid := 1, [159].log_data[5].valid := 1, [159].log_data[6].valid := 1, [159].log_data[7].valid := 1, [159].log_data[8].valid := 1, [159].log_data[9].valid := 1, [159].log_data[10].valid := 1, [159].log_data[11].valid := 1, [159].log_data[12].valid := 1, [159].log_data[13].valid := 1, [159].log_data[14].valid := 1, [159].log_data[15].valid := 1, [159].log_data[16].valid := 1, [159].log_data[17].valid := 1, [159].log_data[18].valid := 1, [159].log_data[19].valid := 1, [159].time.Year := 2023, [159].time.Month := 1, [159].time.Day := 17, [159].time.Hour := 16, [159].time.Minute := 14, [159].time.Second := 59, [160].log_data[0].min := 1.0, [160].log_data[0].max := 1.0, [160].log_data[0].total := 900.0, [160].log_data[0].time := 900.0, [160].log_data[0].minminute := 15, [160].log_data[0].maxminute := 15, [160].log_data[0].valid := 1,
        [160].log_data[1].valid := 1, [160].log_data[2].valid := 1, [160].log_data[3].valid := 1, [160].log_data[4].valid := 1, [160].log_data[5].valid := 1, [160].log_data[6].valid := 1, [160].log_data[7].valid := 1, [160].log_data[8].valid := 1, [160].log_data[9].valid := 1, [160].log_data[10].valid := 1, [160].log_data[11].valid := 1, [160].log_data[12].valid := 1, [160].log_data[13].valid := 1, [160].log_data[14].valid := 1, [160].log_data[15].valid := 1, [160].log_data[16].valid := 1, [160].log_data[17].valid := 1, [160].log_data[18].valid := 1, [160].log_data[19].valid := 1, [160].time.Year := 2023, [160].time.Month := 1, [160].time.Day := 17, [160].time.Hour := 16, [160].time.Minute := 29, [160].time.Second := 59, [161].log_data[0].min := 1.0, [161].log_data[0].max := 1.0, [161].log_data[0].total := 900.0, [161].log_data[0].time := 900.0, [161].log_data[0].minminute := 30, [161].log_data[0].maxminute := 30, [161].log_data[0].valid := 1, [161].log_data[1].valid := 1, [161].log_data[2].valid := 1, [161].log_data[3].valid := 1, [161].log_data[4].valid := 1, [161].log_data[5].valid := 1, [161].log_data[6].valid := 1, [161].log_data[7].valid := 1, [161].log_data[8].valid := 1, [161].log_data[9].valid := 1, [161].log_data[10].valid := 1, [161].log_data[11].valid := 1, [161].log_data[12].valid := 1, [161].log_data[13].valid := 1, [161].log_data[14].valid := 1, [161].log_data[15].valid := 1, [161].log_data[16].valid := 1, [161].log_data[17].valid := 1, [161].log_data[18].valid := 1, [161].log_data[19].valid := 1, [161].time.Year := 2023, [161].time.Month := 1, [161].time.Day := 17, [161].time.Hour := 16, [161].time.Minute := 44, [161].time.Second := 59, [162].log_data[0].min := 1.0, [162].log_data[0].max := 1.0, [162].log_data[0].total := 900.0,
        [162].log_data[0].time := 900.0, [162].log_data[0].minminute := 45, [162].log_data[0].maxminute := 45, [162].log_data[0].valid := 1, [162].log_data[1].valid := 1, [162].log_data[2].valid := 1, [162].log_data[3].valid := 1, [162].log_data[4].valid := 1, [162].log_data[5].valid := 1, [162].log_data[6].valid := 1, [162].log_data[7].valid := 1, [162].log_data[8].valid := 1, [162].log_data[9].valid := 1, [162].log_data[10].valid := 1, [162].log_data[11].valid := 1, [162].log_data[12].valid := 1, [162].log_data[13].valid := 1, [162].log_data[14].valid := 1, [162].log_data[15].valid := 1, [162].log_data[16].valid := 1, [162].log_data[17].valid := 1, [162].log_data[18].valid := 1, [162].log_data[19].valid := 1, [162].time.Year := 2023, [162].time.Month := 1, [162].time.Day := 17, [162].time.Hour := 16, [162].time.Minute := 59, [162].time.Second := 59, [163].log_data[0].min := 1.0, [163].log_data[0].max := 1.0, [163].log_data[0].total := 900.0, [163].log_data[0].time := 900.0, [163].log_data[0].valid := 1, [163].log_data[1].valid := 1, [163].log_data[2].valid := 1, [163].log_data[3].valid := 1, [163].log_data[4].valid := 1, [163].log_data[5].valid := 1, [163].log_data[6].valid := 1, [163].log_data[7].valid := 1, [163].log_data[8].valid := 1, [163].log_data[9].valid := 1, [163].log_data[10].valid := 1, [163].log_data[11].valid := 1, [163].log_data[12].valid := 1, [163].log_data[13].valid := 1, [163].log_data[14].valid := 1, [163].log_data[15].valid := 1, [163].log_data[16].valid := 1, [163].log_data[17].valid := 1, [163].log_data[18].valid := 1, [163].log_data[19].valid := 1, [163].time.Year := 2023, [163].time.Month := 1, [163].time.Day := 17, [163].time.Hour := 17, [163].time.Minute := 14, [163].time.Second := 59, [164].log_data[0].min := 1.0,
        [164].log_data[0].max := 1.0, [164].log_data[0].total := 900.0, [164].log_data[0].time := 900.0, [164].log_data[0].minminute := 15, [164].log_data[0].maxminute := 15, [164].log_data[0].valid := 1, [164].log_data[1].valid := 1, [164].log_data[2].valid := 1, [164].log_data[3].valid := 1, [164].log_data[4].valid := 1, [164].log_data[5].valid := 1, [164].log_data[6].valid := 1, [164].log_data[7].valid := 1, [164].log_data[8].valid := 1, [164].log_data[9].valid := 1, [164].log_data[10].valid := 1, [164].log_data[11].valid := 1, [164].log_data[12].valid := 1, [164].log_data[13].valid := 1, [164].log_data[14].valid := 1, [164].log_data[15].valid := 1, [164].log_data[16].valid := 1, [164].log_data[17].valid := 1, [164].log_data[18].valid := 1, [164].log_data[19].valid := 1, [164].time.Year := 2023, [164].time.Month := 1, [164].time.Day := 17, [164].time.Hour := 17, [164].time.Minute := 29, [164].time.Second := 59, [165].log_data[0].min := 1.0, [165].log_data[0].max := 1.0, [165].log_data[0].total := 900.0, [165].log_data[0].time := 900.0, [165].log_data[0].minminute := 30, [165].log_data[0].maxminute := 30, [165].log_data[0].valid := 1, [165].log_data[1].valid := 1, [165].log_data[2].valid := 1, [165].log_data[3].valid := 1, [165].log_data[4].valid := 1, [165].log_data[5].valid := 1, [165].log_data[6].valid := 1, [165].log_data[7].valid := 1, [165].log_data[8].valid := 1, [165].log_data[9].valid := 1, [165].log_data[10].valid := 1, [165].log_data[11].valid := 1, [165].log_data[12].valid := 1, [165].log_data[13].valid := 1, [165].log_data[14].valid := 1, [165].log_data[15].valid := 1, [165].log_data[16].valid := 1, [165].log_data[17].valid := 1, [165].log_data[18].valid := 1, [165].log_data[19].valid := 1, [165].time.Year := 2023, [165].time.Month := 1, [165].time.Day := 17,
        [165].time.Hour := 17, [165].time.Minute := 44, [165].time.Second := 59, [166].log_data[0].min := 1.0, [166].log_data[0].max := 1.0, [166].log_data[0].total := 900.0, [166].log_data[0].time := 900.0, [166].log_data[0].minminute := 45, [166].log_data[0].maxminute := 45, [166].log_data[0].valid := 1, [166].log_data[1].valid := 1, [166].log_data[2].valid := 1, [166].log_data[3].valid := 1, [166].log_data[4].valid := 1, [166].log_data[5].valid := 1, [166].log_data[6].valid := 1, [166].log_data[7].valid := 1, [166].log_data[8].valid := 1, [166].log_data[9].valid := 1, [166].log_data[10].valid := 1, [166].log_data[11].valid := 1, [166].log_data[12].valid := 1, [166].log_data[13].valid := 1, [166].log_data[14].valid := 1, [166].log_data[15].valid := 1, [166].log_data[16].valid := 1, [166].log_data[17].valid := 1, [166].log_data[18].valid := 1, [166].log_data[19].valid := 1, [166].time.Year := 2023, [166].time.Month := 1, [166].time.Day := 17, [166].time.Hour := 17, [166].time.Minute := 59, [166].time.Second := 59, [167].log_data[0].min := 1.0, [167].log_data[0].max := 1.0, [167].log_data[0].total := 900.0, [167].log_data[0].time := 900.0, [167].log_data[0].valid := 1, [167].log_data[1].valid := 1, [167].log_data[2].valid := 1, [167].log_data[3].valid := 1, [167].log_data[4].valid := 1, [167].log_data[5].valid := 1, [167].log_data[6].valid := 1, [167].log_data[7].valid := 1, [167].log_data[8].valid := 1, [167].log_data[9].valid := 1, [167].log_data[10].valid := 1, [167].log_data[11].valid := 1, [167].log_data[12].valid := 1, [167].log_data[13].valid := 1, [167].log_data[14].valid := 1, [167].log_data[15].valid := 1, [167].log_data[16].valid := 1, [167].log_data[17].valid := 1, [167].log_data[18].valid := 1, [167].log_data[19].valid := 1, [167].time.Year := 2023,
        [167].time.Month := 1, [167].time.Day := 17, [167].time.Hour := 18, [167].time.Minute := 14, [167].time.Second := 59, [168].log_data[0].min := 1.0, [168].log_data[0].max := 1.0, [168].log_data[0].total := 900.0, [168].log_data[0].time := 900.0, [168].log_data[0].minminute := 15, [168].log_data[0].maxminute := 15, [168].log_data[0].valid := 1, [168].log_data[1].valid := 1, [168].log_data[2].valid := 1, [168].log_data[3].valid := 1, [168].log_data[4].valid := 1, [168].log_data[5].valid := 1, [168].log_data[6].valid := 1, [168].log_data[7].valid := 1, [168].log_data[8].valid := 1, [168].log_data[9].valid := 1, [168].log_data[10].valid := 1, [168].log_data[11].valid := 1, [168].log_data[12].valid := 1, [168].log_data[13].valid := 1, [168].log_data[14].valid := 1, [168].log_data[15].valid := 1, [168].log_data[16].valid := 1, [168].log_data[17].valid := 1, [168].log_data[18].valid := 1, [168].log_data[19].valid := 1, [168].time.Year := 2023, [168].time.Month := 1, [168].time.Day := 17, [168].time.Hour := 18, [168].time.Minute := 29, [168].time.Second := 59, [169].log_data[0].min := 1.0, [169].log_data[0].max := 1.0, [169].log_data[0].total := 900.0, [169].log_data[0].time := 900.0, [169].log_data[0].minminute := 30, [169].log_data[0].maxminute := 30, [169].log_data[0].valid := 1, [169].log_data[1].valid := 1, [169].log_data[2].valid := 1, [169].log_data[3].valid := 1, [169].log_data[4].valid := 1, [169].log_data[5].valid := 1, [169].log_data[6].valid := 1, [169].log_data[7].valid := 1, [169].log_data[8].valid := 1, [169].log_data[9].valid := 1, [169].log_data[10].valid := 1, [169].log_data[11].valid := 1, [169].log_data[12].valid := 1, [169].log_data[13].valid := 1, [169].log_data[14].valid := 1, [169].log_data[15].valid := 1, [169].log_data[16].valid := 1,
        [169].log_data[17].valid := 1, [169].log_data[18].valid := 1, [169].log_data[19].valid := 1, [169].time.Year := 2023, [169].time.Month := 1, [169].time.Day := 17, [169].time.Hour := 18, [169].time.Minute := 44, [169].time.Second := 59, [170].log_data[0].min := 1.0, [170].log_data[0].max := 1.0, [170].log_data[0].total := 900.0, [170].log_data[0].time := 900.0, [170].log_data[0].minminute := 45, [170].log_data[0].maxminute := 45, [170].log_data[0].valid := 1, [170].log_data[1].valid := 1, [170].log_data[2].valid := 1, [170].log_data[3].valid := 1, [170].log_data[4].valid := 1, [170].log_data[5].valid := 1, [170].log_data[6].valid := 1, [170].log_data[7].valid := 1, [170].log_data[8].valid := 1, [170].log_data[9].valid := 1, [170].log_data[10].valid := 1, [170].log_data[11].valid := 1, [170].log_data[12].valid := 1, [170].log_data[13].valid := 1, [170].log_data[14].valid := 1, [170].log_data[15].valid := 1, [170].log_data[16].valid := 1, [170].log_data[17].valid := 1, [170].log_data[18].valid := 1, [170].log_data[19].valid := 1, [170].time.Year := 2023, [170].time.Month := 1, [170].time.Day := 17, [170].time.Hour := 18, [170].time.Minute := 59, [170].time.Second := 59, [171].log_data[0].min := 1.0, [171].log_data[0].max := 1.0, [171].log_data[0].total := 900.0, [171].log_data[0].time := 900.0, [171].log_data[0].valid := 1, [171].log_data[1].valid := 1, [171].log_data[2].valid := 1, [171].log_data[3].valid := 1, [171].log_data[4].valid := 1, [171].log_data[5].valid := 1, [171].log_data[6].valid := 1, [171].log_data[7].valid := 1, [171].log_data[8].valid := 1, [171].log_data[9].valid := 1, [171].log_data[10].valid := 1, [171].log_data[11].valid := 1, [171].log_data[12].valid := 1, [171].log_data[13].valid := 1, [171].log_data[14].valid := 1,
        [171].log_data[15].valid := 1, [171].log_data[16].valid := 1, [171].log_data[17].valid := 1, [171].log_data[18].valid := 1, [171].log_data[19].valid := 1, [171].time.Year := 2023, [171].time.Month := 1, [171].time.Day := 17, [171].time.Hour := 19, [171].time.Minute := 14, [171].time.Second := 59, [172].log_data[0].min := 1.0, [172].log_data[0].max := 1.0, [172].log_data[0].total := 900.0, [172].log_data[0].time := 900.0, [172].log_data[0].minminute := 15, [172].log_data[0].maxminute := 15, [172].log_data[0].valid := 1, [172].log_data[1].valid := 1, [172].log_data[2].valid := 1, [172].log_data[3].valid := 1, [172].log_data[4].valid := 1, [172].log_data[5].valid := 1, [172].log_data[6].valid := 1, [172].log_data[7].valid := 1, [172].log_data[8].valid := 1, [172].log_data[9].valid := 1, [172].log_data[10].valid := 1, [172].log_data[11].valid := 1, [172].log_data[12].valid := 1, [172].log_data[13].valid := 1, [172].log_data[14].valid := 1, [172].log_data[15].valid := 1, [172].log_data[16].valid := 1, [172].log_data[17].valid := 1, [172].log_data[18].valid := 1, [172].log_data[19].valid := 1, [172].time.Year := 2023, [172].time.Month := 1, [172].time.Day := 17, [172].time.Hour := 19, [172].time.Minute := 29, [172].time.Second := 59, [173].log_data[0].min := 1.0, [173].log_data[0].max := 1.0, [173].log_data[0].total := 900.0, [173].log_data[0].time := 900.0, [173].log_data[0].minminute := 30, [173].log_data[0].maxminute := 30, [173].log_data[0].valid := 1, [173].log_data[1].valid := 1, [173].log_data[2].valid := 1, [173].log_data[3].valid := 1, [173].log_data[4].valid := 1, [173].log_data[5].valid := 1, [173].log_data[6].valid := 1, [173].log_data[7].valid := 1, [173].log_data[8].valid := 1, [173].log_data[9].valid := 1, [173].log_data[10].valid := 1,
        [173].log_data[11].valid := 1, [173].log_data[12].valid := 1, [173].log_data[13].valid := 1, [173].log_data[14].valid := 1, [173].log_data[15].valid := 1, [173].log_data[16].valid := 1, [173].log_data[17].valid := 1, [173].log_data[18].valid := 1, [173].log_data[19].valid := 1, [173].time.Year := 2023, [173].time.Month := 1, [173].time.Day := 17, [173].time.Hour := 19, [173].time.Minute := 44, [173].time.Second := 59, [174].log_data[0].min := 1.0, [174].log_data[0].max := 1.0, [174].log_data[0].total := 900.0, [174].log_data[0].time := 900.0, [174].log_data[0].minminute := 45, [174].log_data[0].maxminute := 45, [174].log_data[0].valid := 1, [174].log_data[1].valid := 1, [174].log_data[2].valid := 1, [174].log_data[3].valid := 1, [174].log_data[4].valid := 1, [174].log_data[5].valid := 1, [174].log_data[6].valid := 1, [174].log_data[7].valid := 1, [174].log_data[8].valid := 1, [174].log_data[9].valid := 1, [174].log_data[10].valid := 1, [174].log_data[11].valid := 1, [174].log_data[12].valid := 1, [174].log_data[13].valid := 1, [174].log_data[14].valid := 1, [174].log_data[15].valid := 1, [174].log_data[16].valid := 1, [174].log_data[17].valid := 1, [174].log_data[18].valid := 1, [174].log_data[19].valid := 1, [174].time.Year := 2023, [174].time.Month := 1, [174].time.Day := 17, [174].time.Hour := 19, [174].time.Minute := 59, [174].time.Second := 59, [175].log_data[0].min := 1.0, [175].log_data[0].max := 1.0, [175].log_data[0].total := 899.5, [175].log_data[0].time := 899.5, [175].log_data[0].valid := 1, [175].log_data[1].valid := 1, [175].log_data[2].valid := 1, [175].log_data[3].valid := 1, [175].log_data[4].valid := 1, [175].log_data[5].valid := 1, [175].log_data[6].valid := 1, [175].log_data[7].valid := 1, [175].log_data[8].valid := 1,
        [175].log_data[9].valid := 1, [175].log_data[10].valid := 1, [175].log_data[11].valid := 1, [175].log_data[12].valid := 1, [175].log_data[13].valid := 1, [175].log_data[14].valid := 1, [175].log_data[15].valid := 1, [175].log_data[16].valid := 1, [175].log_data[17].valid := 1, [175].log_data[18].valid := 1, [175].log_data[19].valid := 1, [175].time.Year := 2023, [175].time.Month := 1, [175].time.Day := 17, [175].time.Hour := 20, [175].time.Minute := 14, [175].time.Second := 59, [176].log_data[0].min := 1.0, [176].log_data[0].max := 1.0, [176].log_data[0].total := 900.0, [176].log_data[0].time := 900.0, [176].log_data[0].minminute := 15, [176].log_data[0].maxminute := 15, [176].log_data[0].valid := 1, [176].log_data[1].valid := 1, [176].log_data[2].valid := 1, [176].log_data[3].valid := 1, [176].log_data[4].valid := 1, [176].log_data[5].valid := 1, [176].log_data[6].valid := 1, [176].log_data[7].valid := 1, [176].log_data[8].valid := 1, [176].log_data[9].valid := 1, [176].log_data[10].valid := 1, [176].log_data[11].valid := 1, [176].log_data[12].valid := 1, [176].log_data[13].valid := 1, [176].log_data[14].valid := 1, [176].log_data[15].valid := 1, [176].log_data[16].valid := 1, [176].log_data[17].valid := 1, [176].log_data[18].valid := 1, [176].log_data[19].valid := 1, [176].time.Year := 2023, [176].time.Month := 1, [176].time.Day := 17, [176].time.Hour := 20, [176].time.Minute := 29, [176].time.Second := 59, [177].log_data[0].min := 1.0, [177].log_data[0].max := 1.0, [177].log_data[0].total := 900.0, [177].log_data[0].time := 900.0, [177].log_data[0].minminute := 30, [177].log_data[0].maxminute := 30, [177].log_data[0].valid := 1, [177].log_data[1].valid := 1, [177].log_data[2].valid := 1, [177].log_data[3].valid := 1, [177].log_data[4].valid := 1,
        [177].log_data[5].valid := 1, [177].log_data[6].valid := 1, [177].log_data[7].valid := 1, [177].log_data[8].valid := 1, [177].log_data[9].valid := 1, [177].log_data[10].valid := 1, [177].log_data[11].valid := 1, [177].log_data[12].valid := 1, [177].log_data[13].valid := 1, [177].log_data[14].valid := 1, [177].log_data[15].valid := 1, [177].log_data[16].valid := 1, [177].log_data[17].valid := 1, [177].log_data[18].valid := 1, [177].log_data[19].valid := 1, [177].time.Year := 2023, [177].time.Month := 1, [177].time.Day := 17, [177].time.Hour := 20, [177].time.Minute := 44, [177].time.Second := 59, [178].log_data[0].min := 1.0, [178].log_data[0].max := 1.0, [178].log_data[0].total := 900.0, [178].log_data[0].time := 900.0, [178].log_data[0].minminute := 45, [178].log_data[0].maxminute := 45, [178].log_data[0].valid := 1, [178].log_data[1].valid := 1, [178].log_data[2].valid := 1, [178].log_data[3].valid := 1, [178].log_data[4].valid := 1, [178].log_data[5].valid := 1, [178].log_data[6].valid := 1, [178].log_data[7].valid := 1, [178].log_data[8].valid := 1, [178].log_data[9].valid := 1, [178].log_data[10].valid := 1, [178].log_data[11].valid := 1, [178].log_data[12].valid := 1, [178].log_data[13].valid := 1, [178].log_data[14].valid := 1, [178].log_data[15].valid := 1, [178].log_data[16].valid := 1, [178].log_data[17].valid := 1, [178].log_data[18].valid := 1, [178].log_data[19].valid := 1, [178].time.Year := 2023, [178].time.Month := 1, [178].time.Day := 17, [178].time.Hour := 20, [178].time.Minute := 59, [178].time.Second := 59, [179].log_data[0].min := 1.0, [179].log_data[0].max := 1.0, [179].log_data[0].total := 900.0, [179].log_data[0].time := 900.0, [179].log_data[0].valid := 1, [179].log_data[1].valid := 1, [179].log_data[2].valid := 1,
        [179].log_data[3].valid := 1, [179].log_data[4].valid := 1, [179].log_data[5].valid := 1, [179].log_data[6].valid := 1, [179].log_data[7].valid := 1, [179].log_data[8].valid := 1, [179].log_data[9].valid := 1, [179].log_data[10].valid := 1, [179].log_data[11].valid := 1, [179].log_data[12].valid := 1, [179].log_data[13].valid := 1, [179].log_data[14].valid := 1, [179].log_data[15].valid := 1, [179].log_data[16].valid := 1, [179].log_data[17].valid := 1, [179].log_data[18].valid := 1, [179].log_data[19].valid := 1, [179].time.Year := 2023, [179].time.Month := 1, [179].time.Day := 17, [179].time.Hour := 21, [179].time.Minute := 14, [179].time.Second := 59, [180].log_data[0].min := 1.0, [180].log_data[0].max := 1.0, [180].log_data[0].total := 900.0, [180].log_data[0].time := 900.0, [180].log_data[0].minminute := 15, [180].log_data[0].maxminute := 15, [180].log_data[0].valid := 1, [180].log_data[1].valid := 1, [180].log_data[2].valid := 1, [180].log_data[3].valid := 1, [180].log_data[4].valid := 1, [180].log_data[5].valid := 1, [180].log_data[6].valid := 1, [180].log_data[7].valid := 1, [180].log_data[8].valid := 1, [180].log_data[9].valid := 1, [180].log_data[10].valid := 1, [180].log_data[11].valid := 1, [180].log_data[12].valid := 1, [180].log_data[13].valid := 1, [180].log_data[14].valid := 1, [180].log_data[15].valid := 1, [180].log_data[16].valid := 1, [180].log_data[17].valid := 1, [180].log_data[18].valid := 1, [180].log_data[19].valid := 1, [180].time.Year := 2023, [180].time.Month := 1, [180].time.Day := 17, [180].time.Hour := 21, [180].time.Minute := 29, [180].time.Second := 59, [181].log_data[0].min := 1.0, [181].log_data[0].max := 1.0, [181].log_data[0].total := 900.0, [181].log_data[0].time := 900.0, [181].log_data[0].minminute := 30,
        [181].log_data[0].maxminute := 30, [181].log_data[0].valid := 1, [181].log_data[1].valid := 1, [181].log_data[2].valid := 1, [181].log_data[3].valid := 1, [181].log_data[4].valid := 1, [181].log_data[5].valid := 1, [181].log_data[6].valid := 1, [181].log_data[7].valid := 1, [181].log_data[8].valid := 1, [181].log_data[9].valid := 1, [181].log_data[10].valid := 1, [181].log_data[11].valid := 1, [181].log_data[12].valid := 1, [181].log_data[13].valid := 1, [181].log_data[14].valid := 1, [181].log_data[15].valid := 1, [181].log_data[16].valid := 1, [181].log_data[17].valid := 1, [181].log_data[18].valid := 1, [181].log_data[19].valid := 1, [181].time.Year := 2023, [181].time.Month := 1, [181].time.Day := 17, [181].time.Hour := 21, [181].time.Minute := 44, [181].time.Second := 59, [182].log_data[0].min := 1.0, [182].log_data[0].max := 1.0, [182].log_data[0].total := 900.0, [182].log_data[0].time := 900.0, [182].log_data[0].minminute := 45, [182].log_data[0].maxminute := 45, [182].log_data[0].valid := 1, [182].log_data[1].valid := 1, [182].log_data[2].valid := 1, [182].log_data[3].valid := 1, [182].log_data[4].valid := 1, [182].log_data[5].valid := 1, [182].log_data[6].valid := 1, [182].log_data[7].valid := 1, [182].log_data[8].valid := 1, [182].log_data[9].valid := 1, [182].log_data[10].valid := 1, [182].log_data[11].valid := 1, [182].log_data[12].valid := 1, [182].log_data[13].valid := 1, [182].log_data[14].valid := 1, [182].log_data[15].valid := 1, [182].log_data[16].valid := 1, [182].log_data[17].valid := 1, [182].log_data[18].valid := 1, [182].log_data[19].valid := 1, [182].time.Year := 2023, [182].time.Month := 1, [182].time.Day := 17, [182].time.Hour := 21, [182].time.Minute := 59, [182].time.Second := 59, [183].log_data[0].min := 1.0,
        [183].log_data[0].max := 1.0, [183].log_data[0].total := 900.0, [183].log_data[0].time := 900.0, [183].log_data[0].valid := 1, [183].log_data[1].valid := 1, [183].log_data[2].valid := 1, [183].log_data[3].valid := 1, [183].log_data[4].valid := 1, [183].log_data[5].valid := 1, [183].log_data[6].valid := 1, [183].log_data[7].valid := 1, [183].log_data[8].valid := 1, [183].log_data[9].valid := 1, [183].log_data[10].valid := 1, [183].log_data[11].valid := 1, [183].log_data[12].valid := 1, [183].log_data[13].valid := 1, [183].log_data[14].valid := 1, [183].log_data[15].valid := 1, [183].log_data[16].valid := 1, [183].log_data[17].valid := 1, [183].log_data[18].valid := 1, [183].log_data[19].valid := 1, [183].time.Year := 2023, [183].time.Month := 1, [183].time.Day := 17, [183].time.Hour := 22, [183].time.Minute := 14, [183].time.Second := 59, [184].log_data[0].min := 1.0, [184].log_data[0].max := 1.0, [184].log_data[0].total := 900.0, [184].log_data[0].time := 900.0, [184].log_data[0].minminute := 15, [184].log_data[0].maxminute := 15, [184].log_data[0].valid := 1, [184].log_data[1].valid := 1, [184].log_data[2].valid := 1, [184].log_data[3].valid := 1, [184].log_data[4].valid := 1, [184].log_data[5].valid := 1, [184].log_data[6].valid := 1, [184].log_data[7].valid := 1, [184].log_data[8].valid := 1, [184].log_data[9].valid := 1, [184].log_data[10].valid := 1, [184].log_data[11].valid := 1, [184].log_data[12].valid := 1, [184].log_data[13].valid := 1, [184].log_data[14].valid := 1, [184].log_data[15].valid := 1, [184].log_data[16].valid := 1, [184].log_data[17].valid := 1, [184].log_data[18].valid := 1, [184].log_data[19].valid := 1, [184].time.Year := 2023, [184].time.Month := 1, [184].time.Day := 17, [184].time.Hour := 22, [184].time.Minute := 29,
        [184].time.Second := 59, [185].log_data[0].min := 1.0, [185].log_data[0].max := 1.0, [185].log_data[0].total := 900.0, [185].log_data[0].time := 900.0, [185].log_data[0].minminute := 30, [185].log_data[0].maxminute := 30, [185].log_data[0].valid := 1, [185].log_data[1].valid := 1, [185].log_data[2].valid := 1, [185].log_data[3].valid := 1, [185].log_data[4].valid := 1, [185].log_data[5].valid := 1, [185].log_data[6].valid := 1, [185].log_data[7].valid := 1, [185].log_data[8].valid := 1, [185].log_data[9].valid := 1, [185].log_data[10].valid := 1, [185].log_data[11].valid := 1, [185].log_data[12].valid := 1, [185].log_data[13].valid := 1, [185].log_data[14].valid := 1, [185].log_data[15].valid := 1, [185].log_data[16].valid := 1, [185].log_data[17].valid := 1, [185].log_data[18].valid := 1, [185].log_data[19].valid := 1, [185].time.Year := 2023, [185].time.Month := 1, [185].time.Day := 17, [185].time.Hour := 22, [185].time.Minute := 44, [185].time.Second := 59, [186].log_data[0].min := 1.0, [186].log_data[0].max := 1.0, [186].log_data[0].total := 900.0, [186].log_data[0].time := 900.0, [186].log_data[0].minminute := 45, [186].log_data[0].maxminute := 45, [186].log_data[0].valid := 1, [186].log_data[1].valid := 1, [186].log_data[2].valid := 1, [186].log_data[3].valid := 1, [186].log_data[4].valid := 1, [186].log_data[5].valid := 1, [186].log_data[6].valid := 1, [186].log_data[7].valid := 1, [186].log_data[8].valid := 1, [186].log_data[9].valid := 1, [186].log_data[10].valid := 1, [186].log_data[11].valid := 1, [186].log_data[12].valid := 1, [186].log_data[13].valid := 1, [186].log_data[14].valid := 1, [186].log_data[15].valid := 1, [186].log_data[16].valid := 1, [186].log_data[17].valid := 1, [186].log_data[18].valid := 1, [186].log_data[19].valid := 1, [186].time.Year := 2023,
        [186].time.Month := 1, [186].time.Day := 17, [186].time.Hour := 22, [186].time.Minute := 59, [186].time.Second := 59, [187].log_data[0].min := 1.0, [187].log_data[0].max := 1.0, [187].log_data[0].total := 900.0, [187].log_data[0].time := 900.0, [187].log_data[0].valid := 1, [187].log_data[1].valid := 1, [187].log_data[2].valid := 1, [187].log_data[3].valid := 1, [187].log_data[4].valid := 1, [187].log_data[5].valid := 1, [187].log_data[6].valid := 1, [187].log_data[7].valid := 1, [187].log_data[8].valid := 1, [187].log_data[9].valid := 1, [187].log_data[10].valid := 1, [187].log_data[11].valid := 1, [187].log_data[12].valid := 1, [187].log_data[13].valid := 1, [187].log_data[14].valid := 1, [187].log_data[15].valid := 1, [187].log_data[16].valid := 1, [187].log_data[17].valid := 1, [187].log_data[18].valid := 1, [187].log_data[19].valid := 1, [187].time.Year := 2023, [187].time.Month := 1, [187].time.Day := 17, [187].time.Hour := 23, [187].time.Minute := 14, [187].time.Second := 59, [188].log_data[0].min := 1.0, [188].log_data[0].max := 1.0, [188].log_data[0].total := 900.0, [188].log_data[0].time := 900.0, [188].log_data[0].minminute := 15, [188].log_data[0].maxminute := 15, [188].log_data[0].valid := 1, [188].log_data[1].valid := 1, [188].log_data[2].valid := 1, [188].log_data[3].valid := 1, [188].log_data[4].valid := 1, [188].log_data[5].valid := 1, [188].log_data[6].valid := 1, [188].log_data[7].valid := 1, [188].log_data[8].valid := 1, [188].log_data[9].valid := 1, [188].log_data[10].valid := 1, [188].log_data[11].valid := 1, [188].log_data[12].valid := 1, [188].log_data[13].valid := 1, [188].log_data[14].valid := 1, [188].log_data[15].valid := 1, [188].log_data[16].valid := 1, [188].log_data[17].valid := 1, [188].log_data[18].valid := 1,
        [188].log_data[19].valid := 1, [188].time.Year := 2023, [188].time.Month := 1, [188].time.Day := 17, [188].time.Hour := 23, [188].time.Minute := 29, [188].time.Second := 59, [189].log_data[0].min := 1.0, [189].log_data[0].max := 1.0, [189].log_data[0].total := 900.0, [189].log_data[0].time := 900.0, [189].log_data[0].minminute := 30, [189].log_data[0].maxminute := 30, [189].log_data[0].valid := 1, [189].log_data[1].valid := 1, [189].log_data[2].valid := 1, [189].log_data[3].valid := 1, [189].log_data[4].valid := 1, [189].log_data[5].valid := 1, [189].log_data[6].valid := 1, [189].log_data[7].valid := 1, [189].log_data[8].valid := 1, [189].log_data[9].valid := 1, [189].log_data[10].valid := 1, [189].log_data[11].valid := 1, [189].log_data[12].valid := 1, [189].log_data[13].valid := 1, [189].log_data[14].valid := 1, [189].log_data[15].valid := 1, [189].log_data[16].valid := 1, [189].log_data[17].valid := 1, [189].log_data[18].valid := 1, [189].log_data[19].valid := 1, [189].time.Year := 2023, [189].time.Month := 1, [189].time.Day := 17, [189].time.Hour := 23, [189].time.Minute := 44, [189].time.Second := 59, [190].log_data[0].min := 1.0, [190].log_data[0].max := 1.0, [190].log_data[0].total := 900.0, [190].log_data[0].time := 900.0, [190].log_data[0].minminute := 45, [190].log_data[0].maxminute := 45, [190].log_data[0].valid := 1, [190].log_data[1].valid := 1, [190].log_data[2].valid := 1, [190].log_data[3].valid := 1, [190].log_data[4].valid := 1, [190].log_data[5].valid := 1, [190].log_data[6].valid := 1, [190].log_data[7].valid := 1, [190].log_data[8].valid := 1, [190].log_data[9].valid := 1, [190].log_data[10].valid := 1, [190].log_data[11].valid := 1, [190].log_data[12].valid := 1, [190].log_data[13].valid := 1, [190].log_data[14].valid := 1,
        [190].log_data[15].valid := 1, [190].log_data[16].valid := 1, [190].log_data[17].valid := 1, [190].log_data[18].valid := 1, [190].log_data[19].valid := 1, [190].time.Year := 2023, [190].time.Month := 1, [190].time.Day := 17, [190].time.Hour := 23, [190].time.Minute := 59, [190].time.Second := 59, [191].log_data[0].min := 1.0, [191].log_data[0].max := 1.0, [191].log_data[0].total := 900.0, [191].log_data[0].time := 900.0, [191].log_data[0].valid := 1, [191].log_data[1].valid := 1, [191].log_data[2].valid := 1, [191].log_data[3].valid := 1, [191].log_data[4].valid := 1, [191].log_data[5].valid := 1, [191].log_data[6].valid := 1, [191].log_data[7].valid := 1, [191].log_data[8].valid := 1, [191].log_data[9].valid := 1, [191].log_data[10].valid := 1, [191].log_data[11].valid := 1, [191].log_data[12].valid := 1, [191].log_data[13].valid := 1, [191].log_data[14].valid := 1, [191].log_data[15].valid := 1, [191].log_data[16].valid := 1, [191].log_data[17].valid := 1, [191].log_data[18].valid := 1, [191].log_data[19].valid := 1, [191].time.Year := 2023, [191].time.Month := 1, [191].time.Day := 18, [191].time.Minute := 14, [191].time.Second := 59, [192].log_data[0].min := 1.0, [192].log_data[0].max := 1.0, [192].log_data[0].total := 900.0, [192].log_data[0].time := 900.0, [192].log_data[0].minminute := 15, [192].log_data[0].maxminute := 15, [192].log_data[0].valid := 1, [192].log_data[1].valid := 1, [192].log_data[2].valid := 1, [192].log_data[3].valid := 1, [192].log_data[4].valid := 1, [192].log_data[5].valid := 1, [192].log_data[6].valid := 1, [192].log_data[7].valid := 1, [192].log_data[8].valid := 1, [192].log_data[9].valid := 1, [192].log_data[10].valid := 1, [192].log_data[11].valid := 1, [192].log_data[12].valid := 1, [192].log_data[13].valid := 1,
        [192].log_data[14].valid := 1, [192].log_data[15].valid := 1, [192].log_data[16].valid := 1, [192].log_data[17].valid := 1, [192].log_data[18].valid := 1, [192].log_data[19].valid := 1, [192].time.Year := 2023, [192].time.Month := 1, [192].time.Day := 18, [192].time.Minute := 29, [192].time.Second := 59, [193].log_data[0].min := 1.0, [193].log_data[0].max := 1.0, [193].log_data[0].total := 900.0, [193].log_data[0].time := 900.0, [193].log_data[0].minminute := 30, [193].log_data[0].maxminute := 30, [193].log_data[0].valid := 1, [193].log_data[1].valid := 1, [193].log_data[2].valid := 1, [193].log_data[3].valid := 1, [193].log_data[4].valid := 1, [193].log_data[5].valid := 1, [193].log_data[6].valid := 1, [193].log_data[7].valid := 1, [193].log_data[8].valid := 1, [193].log_data[9].valid := 1, [193].log_data[10].valid := 1, [193].log_data[11].valid := 1, [193].log_data[12].valid := 1, [193].log_data[13].valid := 1, [193].log_data[14].valid := 1, [193].log_data[15].valid := 1, [193].log_data[16].valid := 1, [193].log_data[17].valid := 1, [193].log_data[18].valid := 1, [193].log_data[19].valid := 1, [193].time.Year := 2023, [193].time.Month := 1, [193].time.Day := 18, [193].time.Minute := 44, [193].time.Second := 59, [194].log_data[0].min := 1.0, [194].log_data[0].max := 1.0, [194].log_data[0].total := 900.0, [194].log_data[0].time := 900.0, [194].log_data[0].minminute := 45, [194].log_data[0].maxminute := 45, [194].log_data[0].valid := 1, [194].log_data[1].valid := 1, [194].log_data[2].valid := 1, [194].log_data[3].valid := 1, [194].log_data[4].valid := 1, [194].log_data[5].valid := 1, [194].log_data[6].valid := 1, [194].log_data[7].valid := 1, [194].log_data[8].valid := 1, [194].log_data[9].valid := 1, [194].log_data[10].valid := 1, [194].log_data[11].valid := 1,
        [194].log_data[12].valid := 1, [194].log_data[13].valid := 1, [194].log_data[14].valid := 1, [194].log_data[15].valid := 1, [194].log_data[16].valid := 1, [194].log_data[17].valid := 1, [194].log_data[18].valid := 1, [194].log_data[19].valid := 1, [194].time.Year := 2023, [194].time.Month := 1, [194].time.Day := 18, [194].time.Minute := 59, [194].time.Second := 59, [195].log_data[0].min := 1.0, [195].log_data[0].max := 1.0, [195].log_data[0].total := 900.0, [195].log_data[0].time := 900.0, [195].log_data[0].valid := 1, [195].log_data[1].valid := 1, [195].log_data[2].valid := 1, [195].log_data[3].valid := 1, [195].log_data[4].valid := 1, [195].log_data[5].valid := 1, [195].log_data[6].valid := 1, [195].log_data[7].valid := 1, [195].log_data[8].valid := 1, [195].log_data[9].valid := 1, [195].log_data[10].valid := 1, [195].log_data[11].valid := 1, [195].log_data[12].valid := 1, [195].log_data[13].valid := 1, [195].log_data[14].valid := 1, [195].log_data[15].valid := 1, [195].log_data[16].valid := 1, [195].log_data[17].valid := 1, [195].log_data[18].valid := 1, [195].log_data[19].valid := 1, [195].time.Year := 2023, [195].time.Month := 1, [195].time.Day := 18, [195].time.Hour := 1, [195].time.Minute := 14, [195].time.Second := 59, [196].log_data[0].min := 1.0, [196].log_data[0].max := 1.0, [196].log_data[0].total := 900.0, [196].log_data[0].time := 900.0, [196].log_data[0].minminute := 15, [196].log_data[0].maxminute := 15, [196].log_data[0].valid := 1, [196].log_data[1].valid := 1, [196].log_data[2].valid := 1, [196].log_data[3].valid := 1, [196].log_data[4].valid := 1, [196].log_data[5].valid := 1, [196].log_data[6].valid := 1, [196].log_data[7].valid := 1, [196].log_data[8].valid := 1, [196].log_data[9].valid := 1, [196].log_data[10].valid := 1,
        [196].log_data[11].valid := 1, [196].log_data[12].valid := 1, [196].log_data[13].valid := 1, [196].log_data[14].valid := 1, [196].log_data[15].valid := 1, [196].log_data[16].valid := 1, [196].log_data[17].valid := 1, [196].log_data[18].valid := 1, [196].log_data[19].valid := 1, [196].time.Year := 2023, [196].time.Month := 1, [196].time.Day := 18, [196].time.Hour := 1, [196].time.Minute := 29, [196].time.Second := 59, [197].log_data[0].min := 1.0, [197].log_data[0].max := 1.0, [197].log_data[0].total := 900.0, [197].log_data[0].time := 900.0, [197].log_data[0].minminute := 30, [197].log_data[0].maxminute := 30, [197].log_data[0].valid := 1, [197].log_data[1].valid := 1, [197].log_data[2].valid := 1, [197].log_data[3].valid := 1, [197].log_data[4].valid := 1, [197].log_data[5].valid := 1, [197].log_data[6].valid := 1, [197].log_data[7].valid := 1, [197].log_data[8].valid := 1, [197].log_data[9].valid := 1, [197].log_data[10].valid := 1, [197].log_data[11].valid := 1, [197].log_data[12].valid := 1, [197].log_data[13].valid := 1, [197].log_data[14].valid := 1, [197].log_data[15].valid := 1, [197].log_data[16].valid := 1, [197].log_data[17].valid := 1, [197].log_data[18].valid := 1, [197].log_data[19].valid := 1, [197].time.Year := 2023, [197].time.Month := 1, [197].time.Day := 18, [197].time.Hour := 1, [197].time.Minute := 44, [197].time.Second := 59, [198].log_data[0].min := 1.0, [198].log_data[0].max := 1.0, [198].log_data[0].total := 900.0, [198].log_data[0].time := 900.0, [198].log_data[0].minminute := 45, [198].log_data[0].maxminute := 45, [198].log_data[0].valid := 1, [198].log_data[1].valid := 1, [198].log_data[2].valid := 1, [198].log_data[3].valid := 1, [198].log_data[4].valid := 1, [198].log_data[5].valid := 1, [198].log_data[6].valid := 1,
        [198].log_data[7].valid := 1, [198].log_data[8].valid := 1, [198].log_data[9].valid := 1, [198].log_data[10].valid := 1, [198].log_data[11].valid := 1, [198].log_data[12].valid := 1, [198].log_data[13].valid := 1, [198].log_data[14].valid := 1, [198].log_data[15].valid := 1, [198].log_data[16].valid := 1, [198].log_data[17].valid := 1, [198].log_data[18].valid := 1, [198].log_data[19].valid := 1, [198].time.Year := 2023, [198].time.Month := 1, [198].time.Day := 18, [198].time.Hour := 1, [198].time.Minute := 59, [198].time.Second := 59, [199].log_data[0].min := 1.0, [199].log_data[0].max := 1.0, [199].log_data[0].total := 900.0, [199].log_data[0].time := 900.0, [199].log_data[0].valid := 1, [199].log_data[1].valid := 1, [199].log_data[2].valid := 1, [199].log_data[3].valid := 1, [199].log_data[4].valid := 1, [199].log_data[5].valid := 1, [199].log_data[6].valid := 1, [199].log_data[7].valid := 1, [199].log_data[8].valid := 1, [199].log_data[9].valid := 1, [199].log_data[10].valid := 1, [199].log_data[11].valid := 1, [199].log_data[12].valid := 1, [199].log_data[13].valid := 1, [199].log_data[14].valid := 1, [199].log_data[15].valid := 1, [199].log_data[16].valid := 1, [199].log_data[17].valid := 1, [199].log_data[18].valid := 1, [199].log_data[19].valid := 1, [199].time.Year := 2023, [199].time.Month := 1, [199].time.Day := 18, [199].time.Hour := 2, [199].time.Minute := 14, [199].time.Second := 59, [200].log_data[0].min := 1.0, [200].log_data[0].max := 1.0, [200].log_data[0].total := 900.0, [200].log_data[0].time := 900.0, [200].log_data[0].minminute := 15, [200].log_data[0].maxminute := 15, [200].log_data[0].valid := 1, [200].log_data[1].valid := 1, [200].log_data[2].valid := 1, [200].log_data[3].valid := 1, [200].log_data[4].valid := 1,
